    tonFollowerSeq: TON;
	FollowerSeq: SequenceTransfer;	
	lrPosCnt: INT;
	i: INT;
	bRecipeComplete: BOOL;
	rtMasterInRange: R_TRIG;
	bTriggerPos: BOOL;
	tonDelayMotion: TON;
END_VAR

VAR CONSTANT
	iCamID1: MC_CAM_ID:=4;	
    iCamID2: MC_CAM_ID:=5;		
END_VAR

//减速比10/1 同步轮周长400 ，皮带总长3300，7个工位，工位间距60
Ref_MachineStateModel REF= UN01_MachineStateModel;
Ref_Unit REF=Unit01;
ref_Master REF= arVirtualAxisAdmin[1];
ref_Follower1  REF= arRealAxisAdmin[44];
ref_Follower2  REF= arRealAxisAdmin[45];
MainRoution();
CM01_Cam1();
CM02_Cam2();

ACTION Cam1Table:
//凸轮1曲线
camTableFollower1.ArraySize:=SIZEOF(table1);
camTableFollower1.NoOfColumns:=1;
camTableFollower1.NoOfRows:=13;
camTableFollower1.pArray:=ADR(table1);
camTableFollower1.TableType:=MC_TABLETYPE_MOTIONFUNCTION;

{region Table}

//0
table1[1].FunctionType:=MOTIONFUNCTYPE_POLYNOM5;
table1[1].MasterPos:=0;
table1[1].SlavePos:=0;
table1[1].PointIndex:=1;
table1[1].PointType:=MOTIONPOINTTYPE_MOTION;

//1	 (dist200)
table1[2].FunctionType:=MOTIONFUNCTYPE_POLYNOM5;
table1[2].MasterPos:=200;
table1[2].SlavePos:=80;
table1[2].PointIndex:=2;
table1[2].PointType:=MOTIONPOINTTYPE_MOTION;
//2   (dist200)
table1[3].FunctionType:=MOTIONFUNCTYPE_POLYNOM5;
table1[3].MasterPos:=400;
table1[3].SlavePos:=table1[2].SlavePos+60;
table1[3].PointIndex:=3;
table1[3].PointType:=MOTIONPOINTTYPE_MOTION;
//3   (dist200)
table1[4].FunctionType:=MOTIONFUNCTYPE_POLYNOM5;
table1[4].MasterPos:=600;
table1[4].SlavePos:=table1[3].SlavePos+60;
table1[4].PointIndex:=4;
table1[4].PointType:=MOTIONPOINTTYPE_MOTION;
//4  (dist200)
table1[5].FunctionType:=MOTIONFUNCTYPE_POLYNOM5;
table1[5].MasterPos:=800;
table1[5].SlavePos:=table1[4].SlavePos+60;
table1[5].PointIndex:=5;
table1[5].PointType:=MOTIONPOINTTYPE_MOTION;
//5  (dist200)
table1[6].FunctionType:=MOTIONFUNCTYPE_POLYNOM5;
table1[6].MasterPos:=1000;
table1[6].SlavePos:=table1[5].SlavePos+60;
table1[6].PointIndex:=6;
table1[6].PointType:=MOTIONPOINTTYPE_MOTION;
//6  (dist200)
table1[7].FunctionType:=MOTIONFUNCTYPE_POLYNOM5;
table1[7].MasterPos:=1200;
table1[7].SlavePos:=table1[6].SlavePos+60;
table1[7].PointIndex:=7;
table1[7].PointType:=MOTIONPOINTTYPE_MOTION;
//7  (dist200)
table1[8].FunctionType:=MOTIONFUNCTYPE_POLYNOM5;
table1[8].MasterPos:=1400;
table1[8].SlavePos:=table1[7].SlavePos+60;
table1[8].PointIndex:=8;
table1[8].PointType:=MOTIONPOINTTYPE_MOTION;
//900   (dist0)
table1[9].FunctionType:=MOTIONFUNCTYPE_POLYNOM5;
table1[9].MasterPos:=1600;
table1[9].SlavePos:=table1[8].SlavePos+900;
table1[9].PointIndex:=9;
table1[9].PointType:=MOTIONPOINTTYPE_MOTION;
//900  (dist0)
table1[10].FunctionType:=MOTIONFUNCTYPE_POLYNOM5;
table1[10].MasterPos:=1800;
table1[10].SlavePos:=table1[9].SlavePos;
table1[10].PointIndex:=10;
table1[10].PointType:=MOTIONPOINTTYPE_MOTION;
//900  (dist0)
table1[11].FunctionType:=MOTIONFUNCTYPE_POLYNOM5;
table1[11].MasterPos:=2000;
table1[11].SlavePos:=table1[10].SlavePos;
table1[11].PointIndex:=11;
table1[11].PointType:=MOTIONPOINTTYPE_MOTION;
//3240 (dist700)
table1[12].FunctionType:=MOTIONFUNCTYPE_POLYNOM1;
table1[12].MasterPos:=2700;
table1[12].SlavePos:= 3240;
table1[12].PointIndex:=12;
table1[12].PointType:=MOTIONPOINTTYPE_MOTION;
//3300 (dist100)
table1[13].FunctionType:=MOTIONFUNCTYPE_POLYNOM5;
table1[13].MasterPos:=2800;
table1[13].SlavePos:=3300;
table1[13].PointIndex:=13;
table1[13].PointType:=MOTIONPOINTTYPE_MOTION;

{endRegion}
END_ACTION

ACTION Cam1Table_1:
//凸轮1曲线
camTableFollower1.ArraySize:=SIZEOF(table1);
camTableFollower1.NoOfColumns:=1;
camTableFollower1.NoOfRows:=27;
camTableFollower1.pArray:=ADR(table1);
camTableFollower1.TableType:=MC_TABLETYPE_MOTIONFUNCTION;

{region Table}

//0
table1[1].FunctionType:=MOTIONFUNCTYPE_POLYNOM5;
table1[1].MasterPos:=0;
table1[1].SlavePos:=0;
table1[1].PointIndex:=1;
table1[1].PointType:=MOTIONPOINTTYPE_MOTION;

//1	 (dist200)
table1[2].FunctionType:=MOTIONFUNCTYPE_POLYNOM5;
table1[2].MasterPos:=20;
table1[2].SlavePos:=0;
table1[2].PointIndex:=2;
table1[2].PointType:=MOTIONPOINTTYPE_MOTION;

//1	 (dist200)
table1[3].FunctionType:=MOTIONFUNCTYPE_POLYNOM5;
table1[3].MasterPos:=100;
table1[3].SlavePos:=80;
table1[3].PointIndex:=3;
table1[3].PointType:=MOTIONPOINTTYPE_MOTION;
	 
//1	 (dist200)
table1[4].FunctionType:=MOTIONFUNCTYPE_POLYNOM5;
table1[4].MasterPos:=200;
table1[4].SlavePos:=80;
table1[4].PointIndex:=4;
table1[4].PointType:=MOTIONPOINTTYPE_MOTION;
		  
//2   (dist200)
table1[5].FunctionType:=MOTIONFUNCTYPE_POLYNOM5;
table1[5].MasterPos:=220;
table1[5].SlavePos:=80;
table1[5].PointIndex:=5;
table1[5].PointType:=MOTIONPOINTTYPE_MOTION;

//2   (dist200)
table1[6].FunctionType:=MOTIONFUNCTYPE_POLYNOM5;
table1[6].MasterPos:=300;
table1[6].SlavePos:=140;
table1[6].PointIndex:=6;
table1[6].PointType:=MOTIONPOINTTYPE_MOTION;
	 
//2   (dist200)
table1[7].FunctionType:=MOTIONFUNCTYPE_POLYNOM5;
table1[7].MasterPos:=400;
table1[7].SlavePos:=140;
table1[7].PointIndex:=7;
table1[7].PointType:=MOTIONPOINTTYPE_MOTION;

//3   (dist200)
table1[8].FunctionType:=MOTIONFUNCTYPE_POLYNOM5;
table1[8].MasterPos:=420;
table1[8].SlavePos:=200;
table1[8].PointIndex:=8;
table1[8].PointType:=MOTIONPOINTTYPE_MOTION;
		  
//3   (dist200)
table1[9].FunctionType:=MOTIONFUNCTYPE_POLYNOM5;
table1[9].MasterPos:=500;
table1[9].SlavePos:=200;
table1[9].PointIndex:=9;
table1[9].PointType:=MOTIONPOINTTYPE_MOTION;
	 
//3   (dist200)
table1[10].FunctionType:=MOTIONFUNCTYPE_POLYNOM5;
table1[10].MasterPos:=600;
table1[10].SlavePos:=200;
table1[10].PointIndex:=10;
table1[10].PointType:=MOTIONPOINTTYPE_MOTION;		  

//4  (dist200)
table1[11].FunctionType:=MOTIONFUNCTYPE_POLYNOM5;
table1[11].MasterPos:=620;
table1[11].SlavePos:=200;
table1[11].PointIndex:=11;
table1[11].PointType:=MOTIONPOINTTYPE_MOTION;
			   											 
//4  (dist200)
table1[12].FunctionType:=MOTIONFUNCTYPE_POLYNOM5;
table1[12].MasterPos:=700;
table1[12].SlavePos:=260;
table1[12].PointIndex:=12;
table1[12].PointType:=MOTIONPOINTTYPE_MOTION;
	 
//4  (dist200)
table1[13].FunctionType:=MOTIONFUNCTYPE_POLYNOM5;
table1[13].MasterPos:=800;
table1[13].SlavePos:=260;
table1[13].PointIndex:=13;
table1[13].PointType:=MOTIONPOINTTYPE_MOTION;		  
			 
//5  (dist200)
table1[14].FunctionType:=MOTIONFUNCTYPE_POLYNOM5;
table1[14].MasterPos:=820;
table1[14].SlavePos:=260;
table1[14].PointIndex:=14;
table1[14].PointType:=MOTIONPOINTTYPE_MOTION;
  				
//5  (dist200)
table1[15].FunctionType:=MOTIONFUNCTYPE_POLYNOM5;
table1[15].MasterPos:=900;
table1[15].SlavePos:=320;
table1[15].PointIndex:=15;
table1[15].PointType:=MOTIONPOINTTYPE_MOTION;
	 
//5  (dist200)
table1[16].FunctionType:=MOTIONFUNCTYPE_POLYNOM5;
table1[16].MasterPos:=1000;
table1[16].SlavePos:=320;
table1[16].PointIndex:=16;
table1[16].PointType:=MOTIONPOINTTYPE_MOTION;		  
	
//6  (dist200)
table1[17].FunctionType:=MOTIONFUNCTYPE_POLYNOM5;
table1[17].MasterPos:=1020;
table1[17].SlavePos:=320;
table1[17].PointIndex:=17;
table1[17].PointType:=MOTIONPOINTTYPE_MOTION;
		   						  							   
//6  (dist200)
table1[18].FunctionType:=MOTIONFUNCTYPE_POLYNOM5;
table1[18].MasterPos:=1100;
table1[18].SlavePos:=380;
table1[18].PointIndex:=18;
table1[18].PointType:=MOTIONPOINTTYPE_MOTION;
	 
//6  (dist200)
table1[19].FunctionType:=MOTIONFUNCTYPE_POLYNOM5;
table1[19].MasterPos:=1200;
table1[19].SlavePos:=380;
table1[19].PointIndex:=19;
table1[19].PointType:=MOTIONPOINTTYPE_MOTION;		  
	
//7  (dist200)
table1[20].FunctionType:=MOTIONFUNCTYPE_POLYNOM5;
table1[20].MasterPos:=1220;
table1[20].SlavePos:=380;
table1[20].PointIndex:=20;
table1[20].PointType:=MOTIONPOINTTYPE_MOTION;
							 										
//7  (dist200)
table1[21].FunctionType:=MOTIONFUNCTYPE_POLYNOM5;
table1[21].MasterPos:=1300;
table1[21].SlavePos:=440;
table1[21].PointIndex:=21;
table1[21].PointType:=MOTIONPOINTTYPE_MOTION;
	 
//7  (dist200)
table1[22].FunctionType:=MOTIONFUNCTYPE_POLYNOM5;
table1[22].MasterPos:=1400;
table1[22].SlavePos:=440;
table1[22].PointIndex:=22;
table1[22].PointType:=MOTIONPOINTTYPE_MOTION;		  
			   			 
//900   (dist900)
table1[23].FunctionType:=MOTIONFUNCTYPE_POLYNOM5;
table1[23].MasterPos:=1600;
table1[23].SlavePos:=440+900;
table1[23].PointIndex:=23;
table1[23].PointType:=MOTIONPOINTTYPE_MOTION;
//900  (dist0)
table1[24].FunctionType:=MOTIONFUNCTYPE_POLYNOM5;
table1[24].MasterPos:=1900;
table1[24].SlavePos:=1340;
table1[24].PointIndex:=24;
table1[24].PointType:=MOTIONPOINTTYPE_MOTION;
//900  (dist1860)
table1[25].FunctionType:=MOTIONFUNCTYPE_POLYNOM5;
table1[25].MasterPos:=2600;
table1[25].SlavePos:=3200;
table1[25].PointIndex:=25;
table1[25].PointType:=MOTIONPOINTTYPE_MOTION;
//3240 (dist40)
table1[26].FunctionType:=MOTIONFUNCTYPE_POLYNOM1;
table1[26].MasterPos:=2700;
table1[26].SlavePos:= 3240;
table1[26].PointIndex:=26;
table1[26].PointType:=MOTIONPOINTTYPE_MOTION;
//3300 (dist100)
table1[27].FunctionType:=MOTIONFUNCTYPE_POLYNOM5;
table1[27].MasterPos:=2800;
table1[27].SlavePos:=3300;
table1[27].PointIndex:=27;
table1[27].PointType:=MOTIONPOINTTYPE_MOTION;

{endRegion}
END_ACTION

ACTION Cam1Table_2:
//凸轮1曲线
camTableFollower1.ArraySize:=SIZEOF(table1);
camTableFollower1.NoOfColumns:=1;
camTableFollower1.NoOfRows:=20;
camTableFollower1.pArray:=ADR(table1);
camTableFollower1.TableType:=MC_TABLETYPE_MOTIONFUNCTION;

{region Table}

//0
table1[1].FunctionType:=MOTIONFUNCTYPE_POLYNOM5;
table1[1].MasterPos:=0;
table1[1].SlavePos:=0;
table1[1].PointIndex:=1;
table1[1].PointType:=MOTIONPOINTTYPE_MOTION;

//1	 (dist200)
table1[2].FunctionType:=MOTIONFUNCTYPE_POLYNOM5;
table1[2].MasterPos:=100;
table1[2].SlavePos:=80;
table1[2].PointIndex:=2;
table1[2].PointType:=MOTIONPOINTTYPE_MOTION;
	 
//1	 (dist200)
table1[3].FunctionType:=MOTIONFUNCTYPE_POLYNOM5;
table1[3].MasterPos:=200;
table1[3].SlavePos:=80;
table1[3].PointIndex:=3;
table1[3].PointType:=MOTIONPOINTTYPE_MOTION;
		  
//2   (dist200)
table1[4].FunctionType:=MOTIONFUNCTYPE_POLYNOM5;
table1[4].MasterPos:=300;
table1[4].SlavePos:=140;
table1[4].PointIndex:=4;
table1[4].PointType:=MOTIONPOINTTYPE_MOTION;
	 
//2   (dist200)
table1[5].FunctionType:=MOTIONFUNCTYPE_POLYNOM5;
table1[5].MasterPos:=400;
table1[5].SlavePos:=140;
table1[5].PointIndex:=5;
table1[5].PointType:=MOTIONPOINTTYPE_MOTION;

		  
//3   (dist200)
table1[6].FunctionType:=MOTIONFUNCTYPE_POLYNOM5;
table1[6].MasterPos:=500;
table1[6].SlavePos:=200;
table1[6].PointIndex:=6;
table1[6].PointType:=MOTIONPOINTTYPE_MOTION;
	 
//3   (dist200)
table1[7].FunctionType:=MOTIONFUNCTYPE_POLYNOM5;
table1[7].MasterPos:=600;
table1[7].SlavePos:=200;
table1[7].PointIndex:=7;
table1[7].PointType:=MOTIONPOINTTYPE_MOTION;		  
			   											 
//4  (dist200)
table1[8].FunctionType:=MOTIONFUNCTYPE_POLYNOM5;
table1[8].MasterPos:=700;
table1[8].SlavePos:=260;
table1[8].PointIndex:=8;
table1[8].PointType:=MOTIONPOINTTYPE_MOTION;
	 
//4  (dist200)
table1[9].FunctionType:=MOTIONFUNCTYPE_POLYNOM5;
table1[9].MasterPos:=800;
table1[9].SlavePos:=260;
table1[9].PointIndex:=9;
table1[9].PointType:=MOTIONPOINTTYPE_MOTION;		  
			   				
//5  (dist200)
table1[10].FunctionType:=MOTIONFUNCTYPE_POLYNOM5;
table1[10].MasterPos:=900;
table1[10].SlavePos:=320;
table1[10].PointIndex:=10;
table1[10].PointType:=MOTIONPOINTTYPE_MOTION;
	 
//5  (dist200)
table1[11].FunctionType:=MOTIONFUNCTYPE_POLYNOM5;
table1[11].MasterPos:=1000;
table1[11].SlavePos:=320;
table1[11].PointIndex:=11;
table1[11].PointType:=MOTIONPOINTTYPE_MOTION;		  
			   						  							   
//6  (dist200)
table1[12].FunctionType:=MOTIONFUNCTYPE_POLYNOM5;
table1[12].MasterPos:=1100;
table1[12].SlavePos:=380;
table1[12].PointIndex:=12;
table1[12].PointType:=MOTIONPOINTTYPE_MOTION;
	 
//6  (dist200)
table1[13].FunctionType:=MOTIONFUNCTYPE_POLYNOM5;
table1[13].MasterPos:=1200;
table1[13].SlavePos:=380;
table1[13].PointIndex:=13;
table1[13].PointType:=MOTIONPOINTTYPE_MOTION;		  
								 										
//7  (dist200)
table1[14].FunctionType:=MOTIONFUNCTYPE_POLYNOM5;
table1[14].MasterPos:=1300;
table1[14].SlavePos:=440;
table1[14].PointIndex:=14;
table1[14].PointType:=MOTIONPOINTTYPE_MOTION;
	 
//7  (dist200)
table1[15].FunctionType:=MOTIONFUNCTYPE_POLYNOM5;
table1[15].MasterPos:=1400;
table1[15].SlavePos:=440;
table1[15].PointIndex:=15;
table1[15].PointType:=MOTIONPOINTTYPE_MOTION;		  
			   			 
//900   (dist900)
table1[16].FunctionType:=MOTIONFUNCTYPE_POLYNOM5;
table1[16].MasterPos:=1600;
table1[16].SlavePos:=440+900;
table1[16].PointIndex:=16;
table1[16].PointType:=MOTIONPOINTTYPE_MOTION;
//900  (dist0)
table1[17].FunctionType:=MOTIONFUNCTYPE_POLYNOM5;
table1[17].MasterPos:=1900;
table1[17].SlavePos:=1340;
table1[17].PointIndex:=17;
table1[17].PointType:=MOTIONPOINTTYPE_MOTION;
//900  (dist1860)
table1[18].FunctionType:=MOTIONFUNCTYPE_POLYNOM5;
table1[18].MasterPos:=2600;
table1[18].SlavePos:=3200;
table1[18].PointIndex:=18;
table1[18].PointType:=MOTIONPOINTTYPE_MOTION;
//3240 (dist40)
table1[19].FunctionType:=MOTIONFUNCTYPE_POLYNOM1;
table1[19].MasterPos:=2700;
table1[19].SlavePos:= 3240;
table1[19].PointIndex:=19;
table1[19].PointType:=MOTIONPOINTTYPE_MOTION;
//3300 (dist100)
table1[20].FunctionType:=MOTIONFUNCTYPE_POLYNOM5;
table1[20].MasterPos:=2800;
table1[20].SlavePos:=3300;
table1[20].PointIndex:=20;
table1[20].PointType:=MOTIONPOINTTYPE_MOTION;

{endRegion}
END_ACTION

ACTION Cam2Table:
//凸轮2曲线
camTableFollower2.ArraySize:=SIZEOF(table2);
camTableFollower2.NoOfColumns:=1;
camTableFollower2.NoOfRows:=13;
camTableFollower2.pArray:=ADR(table2);
camTableFollower2.TableType:=MC_TABLETYPE_MOTIONFUNCTION;

{region Table}
//7		 							  
table2[1].FunctionType:=MOTIONFUNCTYPE_POLYNOM5;
table2[1].MasterPos:=0;
table2[1].SlavePos:=0;
table2[1].PointIndex:=1;
table2[1].PointType:=MOTIONPOINTTYPE_MOTION;
//900	 (dist300)
table2[2].FunctionType:=MOTIONFUNCTYPE_POLYNOM5;
table2[2].MasterPos:=200;
table2[2].SlavePos:=900;
table2[2].PointIndex:=2;
table2[2].PointType:=MOTIONPOINTTYPE_MOTION;
//900    (dist0)
table2[3].FunctionType:=MOTIONFUNCTYPE_POLYNOM5;
table2[3].MasterPos:=400;
table2[3].SlavePos:=table2[2].SlavePos;
table2[3].PointIndex:=3;
table2[3].PointType:=MOTIONPOINTTYPE_MOTION;
//900    (dist0)
table2[4].FunctionType:=MOTIONFUNCTYPE_POLYNOM5;
table2[4].MasterPos:=600;
table2[4].SlavePos:=table2[3].SlavePos;
table2[4].PointIndex:=4;
table2[4].PointType:=MOTIONPOINTTYPE_MOTION;
//2800 (dist 700)
table2[5].FunctionType:=MOTIONFUNCTYPE_POLYNOM1;
table2[5].MasterPos:=1300;
table2[5].SlavePos:=2800;
table2[5].PointIndex:=5;
table2[5].PointType:=MOTIONPOINTTYPE_MOTION;
//2860 (dist 100)
table2[6].FunctionType:=MOTIONFUNCTYPE_POLYNOM1;
table2[6].MasterPos:=1400;
table2[6].SlavePos:=2860;
table2[6].PointIndex:=6;
table2[6].PointType:=MOTIONPOINTTYPE_MOTION;
//1 (dist 200)
table2[7].FunctionType:=MOTIONFUNCTYPE_POLYNOM5;
table2[7].MasterPos:=1600;
table2[7].SlavePos:=table2[6].SlavePos+80;
table2[7].PointIndex:=7;
table2[7].PointType:=MOTIONPOINTTYPE_MOTION;
//2 (dist 200)
table2[8].FunctionType:=MOTIONFUNCTYPE_POLYNOM5;
table2[8].MasterPos:=1800;
table2[8].SlavePos:=table2[7].SlavePos+60;
table2[8].PointIndex:=8;
table2[8].PointType:=MOTIONPOINTTYPE_MOTION;
//3 (dist 200)
table2[9].FunctionType:=MOTIONFUNCTYPE_POLYNOM5;
table2[9].MasterPos:=2000;
table2[9].SlavePos:=table2[8].SlavePos+60;
table2[9].PointIndex:=9;
table2[9].PointType:=MOTIONPOINTTYPE_MOTION;
//4 (dist 200)
table2[10].FunctionType:=MOTIONFUNCTYPE_POLYNOM5;
table2[10].MasterPos:=2200;
table2[10].SlavePos:=table2[9].SlavePos+60;
table2[10].PointIndex:=10;
table2[10].PointType:=MOTIONPOINTTYPE_MOTION;
//5 (dist 200)
table2[11].FunctionType:=MOTIONFUNCTYPE_POLYNOM5;
table2[11].MasterPos:=2400;
table2[11].SlavePos:=table2[10].SlavePos+60;
table2[11].PointIndex:=11;
table2[11].PointType:=MOTIONPOINTTYPE_MOTION;
//6 (dist 200)
table2[12].FunctionType:=MOTIONFUNCTYPE_POLYNOM5;
table2[12].MasterPos:=2600;
table2[12].SlavePos:=table2[11].SlavePos+60;
table2[12].PointIndex:=12;
table2[12].PointType:=MOTIONPOINTTYPE_MOTION;
//7 (dist 200)
table2[13].FunctionType:=MOTIONFUNCTYPE_POLYNOM5;
table2[13].MasterPos:=2800;
table2[13].SlavePos:=3300;
table2[13].PointIndex:=13;
table2[13].PointType:=MOTIONPOINTTYPE_MOTION;

{endRegion}
END_ACTION

ACTION Cam2Table_1:
//凸轮2曲线
camTableFollower2.ArraySize:=SIZEOF(table2);
camTableFollower2.NoOfColumns:=1;
camTableFollower2.NoOfRows:=27;
camTableFollower2.pArray:=ADR(table2);
camTableFollower2.TableType:=MC_TABLETYPE_MOTIONFUNCTION;

{region Table}
//7		 							  
table2[1].FunctionType:=MOTIONFUNCTYPE_POLYNOM5;
table2[1].MasterPos:=0;
table2[1].SlavePos:=0;
table2[1].PointIndex:=1;
table2[1].PointType:=MOTIONPOINTTYPE_MOTION;
	 
//900	 (dist900)
table2[2].FunctionType:=MOTIONFUNCTYPE_POLYNOM5;
table2[2].MasterPos:=200;
table2[2].SlavePos:=900;
table2[2].PointIndex:=2;
table2[2].PointType:=MOTIONPOINTTYPE_MOTION;
	 
//900    (dist0)
table2[3].FunctionType:=MOTIONFUNCTYPE_POLYNOM5;
table2[3].MasterPos:=500;
table2[3].SlavePos:=900;
table2[3].PointIndex:=3;
table2[3].PointType:=MOTIONPOINTTYPE_MOTION;
//900    (dist1860)
table2[4].FunctionType:=MOTIONFUNCTYPE_POLYNOM5;
table2[4].MasterPos:=1200;
table2[4].SlavePos:=2760;
table2[4].PointIndex:=4;
table2[4].PointType:=MOTIONPOINTTYPE_MOTION;
	 
//2800 (dist 40)
table2[5].FunctionType:=MOTIONFUNCTYPE_POLYNOM1;
table2[5].MasterPos:=1300;
table2[5].SlavePos:=2800;
table2[5].PointIndex:=5;
table2[5].PointType:=MOTIONPOINTTYPE_MOTION;
	 
//2860 (dist 100)
table2[6].FunctionType:=MOTIONFUNCTYPE_POLYNOM1;
table2[6].MasterPos:=1400;
table2[6].SlavePos:=2860;
table2[6].PointIndex:=6;
table2[6].PointType:=MOTIONPOINTTYPE_MOTION;
	 
//1 (dist 200)
table2[7].FunctionType:=MOTIONFUNCTYPE_POLYNOM5;
table2[7].MasterPos:=1420;
table2[7].SlavePos:=2860;
table2[7].PointIndex:=7;
table2[7].PointType:=MOTIONPOINTTYPE_MOTION;		  
			   
//1 (dist 200)
table2[8].FunctionType:=MOTIONFUNCTYPE_POLYNOM5;
table2[8].MasterPos:=1500;
table2[8].SlavePos:=2940;
table2[8].PointIndex:=8;
table2[8].PointType:=MOTIONPOINTTYPE_MOTION;
	 
//1 (dist 200)
table2[9].FunctionType:=MOTIONFUNCTYPE_POLYNOM5;
table2[9].MasterPos:=1600;
table2[9].SlavePos:=2940;
table2[9].PointIndex:=9;
table2[9].PointType:=MOTIONPOINTTYPE_MOTION;

//2 (dist 200)
table2[10].FunctionType:=MOTIONFUNCTYPE_POLYNOM5;
table2[10].MasterPos:=1620;
table2[10].SlavePos:=2940;
table2[10].PointIndex:=10;
table2[10].PointType:=MOTIONPOINTTYPE_MOTION;
	 
//2 (dist 200)
table2[11].FunctionType:=MOTIONFUNCTYPE_POLYNOM5;
table2[11].MasterPos:=1700;
table2[11].SlavePos:=3000;
table2[11].PointIndex:=11;
table2[11].PointType:=MOTIONPOINTTYPE_MOTION;
	 
//2 (dist 200)
table2[12].FunctionType:=MOTIONFUNCTYPE_POLYNOM5;
table2[12].MasterPos:=1800;
table2[12].SlavePos:=3000;
table2[12].PointIndex:=12;
table2[12].PointType:=MOTIONPOINTTYPE_MOTION;
	
//3 (dist 200)
table2[13].FunctionType:=MOTIONFUNCTYPE_POLYNOM5;
table2[13].MasterPos:=1820;
table2[13].SlavePos:=3000;
table2[13].PointIndex:=13;
table2[13].PointType:=MOTIONPOINTTYPE_MOTION;
 
//3 (dist 200)
table2[14].FunctionType:=MOTIONFUNCTYPE_POLYNOM5;
table2[14].MasterPos:=1900;
table2[14].SlavePos:=3060;
table2[14].PointIndex:=14;
table2[14].PointType:=MOTIONPOINTTYPE_MOTION;
	 
//3 (dist 200)
table2[15].FunctionType:=MOTIONFUNCTYPE_POLYNOM5;
table2[15].MasterPos:=2000;
table2[15].SlavePos:=3060;
table2[15].PointIndex:=15;
table2[15].PointType:=MOTIONPOINTTYPE_MOTION;
	  
//4 (dist 200)
table2[16].FunctionType:=MOTIONFUNCTYPE_POLYNOM5;
table2[16].MasterPos:=2020;
table2[16].SlavePos:=3060;
table2[16].PointIndex:=16;
table2[16].PointType:=MOTIONPOINTTYPE_MOTION;
	 
//4 (dist 200)
table2[17].FunctionType:=MOTIONFUNCTYPE_POLYNOM5;
table2[17].MasterPos:=2100;
table2[17].SlavePos:=3120;
table2[17].PointIndex:=17;
table2[17].PointType:=MOTIONPOINTTYPE_MOTION;		  
			   
//4 (dist 200)
table2[18].FunctionType:=MOTIONFUNCTYPE_POLYNOM5;
table2[18].MasterPos:=2200;
table2[18].SlavePos:=3120;
table2[18].PointIndex:=18;
table2[18].PointType:=MOTIONPOINTTYPE_MOTION;
	 
//5 (dist 200)
table2[19].FunctionType:=MOTIONFUNCTYPE_POLYNOM5;
table2[19].MasterPos:=2220;
table2[19].SlavePos:=3120;
table2[19].PointIndex:=19;
table2[19].PointType:=MOTIONPOINTTYPE_MOTION;
	 
//5 (dist 200)
table2[20].FunctionType:=MOTIONFUNCTYPE_POLYNOM5;
table2[20].MasterPos:=2300;
table2[20].SlavePos:=3180;
table2[20].PointIndex:=20;
table2[20].PointType:=MOTIONPOINTTYPE_MOTION;
		  
//5 (dist 200)
table2[21].FunctionType:=MOTIONFUNCTYPE_POLYNOM5;
table2[21].MasterPos:=2400;
table2[21].SlavePos:=3180;
table2[21].PointIndex:=21;
table2[21].PointType:=MOTIONPOINTTYPE_MOTION;	 
	 
//6 (dist 200)
table2[22].FunctionType:=MOTIONFUNCTYPE_POLYNOM5;
table2[22].MasterPos:=2420;
table2[22].SlavePos:=3180;
table2[22].PointIndex:=22;
table2[22].PointType:=MOTIONPOINTTYPE_MOTION;
		  
//6 (dist 200)
table2[23].FunctionType:=MOTIONFUNCTYPE_POLYNOM5;
table2[23].MasterPos:=2500;
table2[23].SlavePos:=3240;
table2[23].PointIndex:=23;
table2[23].PointType:=MOTIONPOINTTYPE_MOTION;

//6 (dist 200)
table2[24].FunctionType:=MOTIONFUNCTYPE_POLYNOM5;
table2[24].MasterPos:=2600;
table2[24].SlavePos:=3240;
table2[24].PointIndex:=24;
table2[24].PointType:=MOTIONPOINTTYPE_MOTION;	 
		  	   
//7 (dist 200)
table2[25].FunctionType:=MOTIONFUNCTYPE_POLYNOM5;
table2[25].MasterPos:=2620;
table2[25].SlavePos:=3240;
table2[25].PointIndex:=25;
table2[25].PointType:=MOTIONPOINTTYPE_MOTION;

//7 (dist 200)
table2[26].FunctionType:=MOTIONFUNCTYPE_POLYNOM5;
table2[26].MasterPos:=2700;
table2[26].SlavePos:=3300;
table2[26].PointIndex:=26;
table2[26].PointType:=MOTIONPOINTTYPE_MOTION;	 
		  
//7 (dist 200)
table2[27].FunctionType:=MOTIONFUNCTYPE_POLYNOM5;
table2[27].MasterPos:=2800;
table2[27].SlavePos:=3300;
table2[27].PointIndex:=27;
table2[27].PointType:=MOTIONPOINTTYPE_MOTION;
	 
{endRegion}
END_ACTION

ACTION Cam2Table_2:
//凸轮2曲线
camTableFollower2.ArraySize:=SIZEOF(table2);
camTableFollower2.NoOfColumns:=1;
camTableFollower2.NoOfRows:=20;
camTableFollower2.pArray:=ADR(table2);
camTableFollower2.TableType:=MC_TABLETYPE_MOTIONFUNCTION;

{region Table}
//7		 							  
table2[1].FunctionType:=MOTIONFUNCTYPE_POLYNOM5;
table2[1].MasterPos:=0;
table2[1].SlavePos:=0;
table2[1].PointIndex:=1;
table2[1].PointType:=MOTIONPOINTTYPE_MOTION;
//900	 (dist900)
table2[2].FunctionType:=MOTIONFUNCTYPE_POLYNOM5;
table2[2].MasterPos:=200;
table2[2].SlavePos:=900;
table2[2].PointIndex:=2;
table2[2].PointType:=MOTIONPOINTTYPE_MOTION;
//900    (dist0)
table2[3].FunctionType:=MOTIONFUNCTYPE_POLYNOM5;
table2[3].MasterPos:=500;
table2[3].SlavePos:=900;
table2[3].PointIndex:=3;
table2[3].PointType:=MOTIONPOINTTYPE_MOTION;
//900    (dist1860)
table2[4].FunctionType:=MOTIONFUNCTYPE_POLYNOM5;
table2[4].MasterPos:=1200;
table2[4].SlavePos:=2760;
table2[4].PointIndex:=4;
table2[4].PointType:=MOTIONPOINTTYPE_MOTION;
//2800 (dist 40)
table2[5].FunctionType:=MOTIONFUNCTYPE_POLYNOM1;
table2[5].MasterPos:=1300;
table2[5].SlavePos:=2800;
table2[5].PointIndex:=5;
table2[5].PointType:=MOTIONPOINTTYPE_MOTION;
//2860 (dist 100)
table2[6].FunctionType:=MOTIONFUNCTYPE_POLYNOM1;
table2[6].MasterPos:=1400;
table2[6].SlavePos:=2860;
table2[6].PointIndex:=6;
table2[6].PointType:=MOTIONPOINTTYPE_MOTION;
//1 (dist 200)
table2[7].FunctionType:=MOTIONFUNCTYPE_POLYNOM5;
table2[7].MasterPos:=1500;
table2[7].SlavePos:=2940;
table2[7].PointIndex:=7;
table2[7].PointType:=MOTIONPOINTTYPE_MOTION;
//1 (dist 200)
table2[8].FunctionType:=MOTIONFUNCTYPE_POLYNOM5;
table2[8].MasterPos:=1600;
table2[8].SlavePos:=2940;
table2[8].PointIndex:=8;
table2[8].PointType:=MOTIONPOINTTYPE_MOTION;
	 
//2 (dist 200)
table2[9].FunctionType:=MOTIONFUNCTYPE_POLYNOM5;
table2[9].MasterPos:=1700;
table2[9].SlavePos:=3000;
table2[9].PointIndex:=9;
table2[9].PointType:=MOTIONPOINTTYPE_MOTION;
//2 (dist 200)
table2[10].FunctionType:=MOTIONFUNCTYPE_POLYNOM5;
table2[10].MasterPos:=1800;
table2[10].SlavePos:=3000;
table2[10].PointIndex:=10;
table2[10].PointType:=MOTIONPOINTTYPE_MOTION;
	 
//3 (dist 200)
table2[11].FunctionType:=MOTIONFUNCTYPE_POLYNOM5;
table2[11].MasterPos:=1900;
table2[11].SlavePos:=3060;
table2[11].PointIndex:=11;
table2[11].PointType:=MOTIONPOINTTYPE_MOTION;
//3 (dist 200)
table2[12].FunctionType:=MOTIONFUNCTYPE_POLYNOM5;
table2[12].MasterPos:=2000;
table2[12].SlavePos:=3060;
table2[12].PointIndex:=12;
table2[12].PointType:=MOTIONPOINTTYPE_MOTION;
	  
//4 (dist 200)
table2[13].FunctionType:=MOTIONFUNCTYPE_POLYNOM5;
table2[13].MasterPos:=2100;
table2[13].SlavePos:=3120;
table2[13].PointIndex:=13;
table2[13].PointType:=MOTIONPOINTTYPE_MOTION;
//4 (dist 200)
table2[14].FunctionType:=MOTIONFUNCTYPE_POLYNOM5;
table2[14].MasterPos:=2200;
table2[14].SlavePos:=3120;
table2[14].PointIndex:=14;
table2[14].PointType:=MOTIONPOINTTYPE_MOTION;
	 
//5 (dist 200)
table2[15].FunctionType:=MOTIONFUNCTYPE_POLYNOM5;
table2[15].MasterPos:=2300;
table2[15].SlavePos:=3180;
table2[15].PointIndex:=15;
table2[15].PointType:=MOTIONPOINTTYPE_MOTION;
//5 (dist 200)
table2[16].FunctionType:=MOTIONFUNCTYPE_POLYNOM5;
table2[16].MasterPos:=2400;
table2[16].SlavePos:=3180;
table2[16].PointIndex:=16;
table2[16].PointType:=MOTIONPOINTTYPE_MOTION;	 
	 
//6 (dist 200)
table2[17].FunctionType:=MOTIONFUNCTYPE_POLYNOM5;
table2[17].MasterPos:=2500;
table2[17].SlavePos:=3240;
table2[17].PointIndex:=17;
table2[17].PointType:=MOTIONPOINTTYPE_MOTION;

//6 (dist 200)
table2[18].FunctionType:=MOTIONFUNCTYPE_POLYNOM5;
table2[18].MasterPos:=2600;
table2[18].SlavePos:=3240;
table2[18].PointIndex:=18;
table2[18].PointType:=MOTIONPOINTTYPE_MOTION;	 
		  	   
//7 (dist 200)
table2[19].FunctionType:=MOTIONFUNCTYPE_POLYNOM5;
table2[19].MasterPos:=2700;
table2[19].SlavePos:=3300;
table2[19].PointIndex:=19;
table2[19].PointType:=MOTIONPOINTTYPE_MOTION;
//7 (dist 200)
table2[20].FunctionType:=MOTIONFUNCTYPE_POLYNOM5;
table2[20].MasterPos:=2800;
table2[20].SlavePos:=3300;
table2[20].PointIndex:=20;
table2[20].PointType:=MOTIONPOINTTYPE_MOTION;
	 
{endRegion}
END_ACTION

ACTION CM01_Cam1:
Cam1Table();
	 
MC_CamIn_Follower1.Scaling.MasterRelative:=FALSE;
MC_CamIn_Follower1.Scaling.SlaveRelative:=FALSE;	 
	 
MC_CamIn_Follower1(
	Master:=ref_Master.Axis , 
	Slave:= ref_Follower1.Axis, 
	Execute:= ref_Follower1.i.CamIn, 
	ActivationMode:= , 
	ActivationPosition:= , 
	CamTableID:=iCamID1 , 
	Scaling:= , 
	Options:= , 
	InSync=> ref_Follower1.o.InCam, 
	Busy=> , 
	Active=> , 
	CommandAborted=> , 
	Error=> , 
	ErrorID=> );	
	
MC_CamTableSelect_Follower1(
	Master:= ref_Master.Axis, 
	Slave:= ref_Follower1.Axis, 
	CamTable:= CamTableFollower1, 
	Execute:= ref_Follower1.i.SelectCamTable, 
	Periodic:= TRUE, 
	MasterAbsolute:= , 
	SlaveAbsolute:= , 
	CamTableID:= iCamID1, 
	Done=> ref_Follower1.o.SelectCamTableDone, 
	Busy=> , 
	Error=> , 
	ErrorID=> );


MC_GearIn_Follower1(
	Master:=ref_Follower2.Axis , 
	Slave:=ref_Follower1.Axis , 
	Execute:=ref_Follower1.i.GearIn , 
	RatioNumerator:= 1, 
	RatioDenominator:= 1, 
	Acceleration:= , 
	Deceleration:= , 
	Jerk:= , 
	BufferMode:= , 
	Options:= , 
	InGear=> ref_Follower1.o.InGear, 
	Busy=> , 
	Active=> , 
	CommandAborted=> , 
	Error=> , 
	ErrorID=> );	
	
MC_ReadCamTableSlaveDynamicsFollwer1(
	Execute:= , 
	CamTableID:= iCamID1, 
	MasterPosition:= ref_Master.o.ActPos, 
	Done=> , 
	Busy=> , 
	Error=> , 
	ErrorID=> , 
	SlavePosition=> , 
	SlaveVelocity=> , 
	SlaveAcceleration=> );
END_ACTION

ACTION CM02_Cam2:
Cam2Table();

MC_CamIn_Follower2.Scaling.MasterRelative:=FALSE;
MC_CamIn_Follower2.Scaling.SlaveRelative:=FALSE;		 
MC_CamIn_Follower2(
	Master:=ref_Master.Axis , 
	Slave:= ref_Follower2.Axis, 
	Execute:= ref_Follower2.i.CamIn, 
	ActivationMode:= , 
	ActivationPosition:= , 
	CamTableID:=iCamID2 , 
	Scaling:= , 
	Options:= , 
	InSync=> ref_Follower2.o.InCam, 
	Busy=> , 
	Active=> , 
	CommandAborted=> , 
	Error=> , 
	ErrorID=> );	
	
MC_CamTableSelect_Follower2(
	Master:= ref_Master.Axis, 
	Slave:= ref_Follower2.Axis, 
	CamTable:= CamTableFollower2, 
	Execute:= ref_Follower2.i.SelectCamTable, 
	Periodic:= TRUE, 
	MasterAbsolute:= , 
	SlaveAbsolute:= , 
	CamTableID:= iCamID2, 
	Done=> ref_Follower2.o.SelectCamTableDone, 
	Busy=> , 
	Error=> , 
	ErrorID=> );

MC_GearIn_Follower2(
	Master:=ref_Follower1.Axis , 
	Slave:=ref_Follower2.Axis , 
	Execute:=ref_Follower2.i.GearIn , 
	RatioNumerator:= 1, 
	RatioDenominator:= 1, 
	Acceleration:= , 
	Deceleration:= , 
	Jerk:= , 
	BufferMode:= , 
	Options:= , 
	InGear=> ref_Follower2.o.InGear, 
	Busy=> , 
	Active=> , 
	CommandAborted=> , 
	Error=> , 
	ErrorID=> );		
	
	
MC_ReadCamTableSlaveDynamicsFollwer2(
	Execute:= , 
	CamTableID:= iCamID2, 
	MasterPosition:= ref_Master.o.ActPos, 
	Done=> , 
	Busy=> , 
	Error=> , 
	ErrorID=> , 
	SlavePosition=> , 
	SlaveVelocity=> , 
	SlaveAcceleration=> );
END_ACTION

ACTION CM03_Follower:
CASE FollowerSeq.Now OF
	0: 
	   IF Ref_MachineStateModel.Sts_Resetting THEN
		  FollowerSeq(ExeCute:= TRUE, Next:= Seq_Resetting);  
	   END_IF	
	   IF Ref_MachineStateModel.Sts_Stopping  THEN
		  FollowerSeq(ExeCute:= TRUE, Next:= Seq_Stopping);  
	   END_IF
	   IF Ref_MachineStateModel.Sts_Execute  THEN
		  FollowerSeq(ExeCute:= TRUE, Next:= 110);   
	   END_IF
{region Resetting} 
	10:
		IF NOT ref_Follower1.o.PowerOn  THEN;
		   ref_Follower1.i.Enable:=TRUE;
		END_IF
		IF NOT ref_Follower2.o.PowerOn  THEN;
		   ref_Follower2.i.Enable:=TRUE;
		END_IF	
		
		IF ref_Follower1.o.PowerOn AND ref_Follower2.o.PowerOn THEN
		   FollowerSeq(ExeCute:= TRUE, Next:= 20);  
		END_IF
        IF Ref_MachineStateModel.Sts_Stopping  THEN
		   FollowerSeq(ExeCute:= TRUE, Next:= Seq_Stopping);  
	    END_IF	
		
	20:
		IF glb_AllAxisHomed_UN01 THEN
		   FollowerSeq(ExeCute:= TRUE, Next:= 21);
		   ELSE 
		   FollowerSeq(ExeCute:= TRUE, Next:= 30);
		END_IF
		
	21:
		IF ref_Master.o.Homed AND ref_Master.o.PowerOn THEN
		   FollowerSeq(ExeCute:= TRUE, Next:= 60);//轴组耦合
		END_IF
	30:
	   glb_lrMasterWrkCnt:=0;
	   glb_lrMasterTargetCnt:=0;
	   bRecipeComplete:=FALSE;
       MEMSET(destAddr:= ADR(glb_BinBelt4_5), fillByte:= 0, n:= SIZEOF(glb_BinBelt4_5));      
	   FollowerSeq(ExeCute:= TRUE, Next:= 40);
	
	40: 
	   ref_Follower1.i.GearIn:=TRUE;
	   IF ref_Follower1.o.InGear THEN
		  FollowerSeq(ExeCute:= TRUE, Next:= 41);
	   END_IF
	   
	41:
       ref_Follower2.i.HomeMode:=0;
       ref_Follower2.i.HomeOffset:=290;  //	
	   tonFollowerSeq(IN:=TRUE , PT:=T#1S , Q=> , ET=> );
	   IF tonFollowerSeq.Q THEN
		  tonFollowerSeq(IN:=FALSE , PT:=T#1S , Q=> , ET=> );	   
			ref_Follower2.i.Home:=TRUE;
			FollowerSeq(ExeCute:= TRUE, Next:= 42);
	   END_IF
	   
	42:
       IF ref_Follower2.o.HomeDone THEN
		  ref_Follower2.i.Home:=FALSE;
		  FollowerSeq(ExeCute:= TRUE, Next:= 43); 
	   ELSE IF Ref_MachineStateModel.Sts_Stopping  THEN
		       ref_Follower2.i.Home:=FALSE;
               FollowerSeq(ExeCute:= TRUE, Next:= Seq_Stopping);
	        END_IF
	   END_IF
	   
	43:
	   ref_Follower1.i.GearOut:=TRUE;
	   IF ref_Follower1.o.GearOutDone AND NOT ref_Follower1.o.InSync THEN
		  ref_Follower1.i.GearOut:=FALSE;
		  ref_Follower1.i.GearIn:=FALSE;
		  FollowerSeq(ExeCute:= TRUE, Next:= 44); 
	   END_IF
	   
	44:
	   IF ref_Follower1.o.StandStill THEN
          FollowerSeq(ExeCute:= TRUE, Next:= 45);
	   ELSE IF Ref_MachineStateModel.Sts_Stopping  THEN
		       FollowerSeq(ExeCute:= TRUE, Next:= Seq_Stopping);   
		    END_IF	  
	   END_IF
	   
	45:
	   ref_Follower2.i.GearIn:=TRUE;
	   IF ref_Follower2.o.InGear THEN
		  FollowerSeq(ExeCute:= TRUE, Next:= 46); 
	   END_IF  
	46:
	      ref_Follower1.i.HomeOffset:=290; // 
	      tonFollowerSeq(IN:=TRUE , PT:=T#1S , Q=> , ET=> );
	   IF tonFollowerSeq.Q THEN
			tonFollowerSeq(IN:=FALSE , PT:=T#1S , Q=> , ET=> );	   
			ref_Follower1.i.Home:=TRUE;
			FollowerSeq(ExeCute:= TRUE, Next:= 47); 
	   END_IF
	   
	47:
       IF ref_Follower1.o.HomeDone THEN
		   ref_Follower1.i.Home:=FALSE;
		   FollowerSeq(ExeCute:= TRUE, Next:= 48);
	   ELSE IF Ref_MachineStateModel.Sts_Stopping  THEN
		       ref_Follower1.i.Home:=FALSE;
               FollowerSeq(ExeCute:= TRUE, Next:= Seq_Stopping);   
		    END_IF 
	   END_IF
	48:
    	 ref_Follower1.i.Pos:=0 ; 
	     ref_Follower1.i.Vel:=100;
	     ref_Follower1.i.Acc:=600;
	     ref_Follower1.i.Dec:=600;   
		 FollowerSeq(ExeCute:= TRUE, Next:= 49);
    49: 
		 ref_Follower1.i.MoveAbs:=TRUE;
	     IF  ref_Follower1.o.CmdDone  THEN
			 ref_Follower1.i.MoveAbs:=FALSE; 
			 FollowerSeq(ExeCute:= TRUE, Next:= 50);
	     ELSE IF Ref_MachineStateModel.Sts_Stopping  THEN
		         ref_Follower1.i.MoveAbs:=FALSE;
                 FollowerSeq(ExeCute:= TRUE, Next:= Seq_Stopping);   
		      END_IF			 
		 END_IF
	      
	50:
	   ref_Follower2.i.GearOut:=TRUE;
	   IF ref_Follower2.o.GearOutDone  THEN
		  ref_Follower2.i.GearOut:=FALSE;
		  ref_Follower2.i.GearIn:=FALSE;
		  FollowerSeq(ExeCute:= TRUE, Next:= 51); 
	   END_IF  
	51: 
        tonFollowerSeq(IN:=TRUE , PT:=T#500MS , Q=> , ET=> );
		IF  ref_Follower2.o.StandStill AND tonFollowerSeq.Q  THEN
			 tonFollowerSeq(IN:=FALSE , PT:=T#500MS , Q=> , ET=> );
		     FollowerSeq(ExeCute:= TRUE, Next:= 52);
	    END_IF
		
	52: 
		 ref_Follower2.i.Dist:=440-ref_Follower2.o.ActPos ; 
         lrFollower2PosLast:=ref_Follower2.i.Pos;
	     ref_Follower2.i.Vel:=100;
	     ref_Follower2.i.Acc:=6000;
	     ref_Follower2.i.Dec:=600;
		 FollowerSeq(ExeCute:= TRUE, Next:= 53);
		 
    53:  ref_Follower2.i.MoveReal:=TRUE; 
		 FollowerSeq(ExeCute:= TRUE, Next:= 54);

    54:		 
         IF  ref_Follower2.o.CmdDone  THEN
			 ref_Follower2.i.MoveReal:=FALSE; 
			 FollowerSeq(ExeCute:= TRUE, Next:= 55);
	     ELSE IF Ref_MachineStateModel.Sts_Stopping  THEN
                 FollowerSeq(ExeCute:= TRUE, Next:= Seq_Stopping);    
		      END_IF			 
		 END_IF
    55: 		 
	   ref_Follower2.i.Home:=TRUE;
	   ref_Follower2.i.HomeOffset:=0;  
	   ref_Follower2.i.HomeMode:=2;
	   FollowerSeq(ExeCute:= TRUE, Next:= 56); 
	   
	56:
       IF ref_Follower2.o.HomeDone THEN
		   ref_Follower2.i.Home:=FALSE;
		   FollowerSeq(ExeCute:= TRUE, Next:= 60);  
	   ELSE IF Ref_MachineStateModel.Sts_Stopping  THEN
		       FollowerSeq(ExeCute:= TRUE, Next:= Seq_Stopping);   
		    END_IF		   
	   END_IF
	   
	60:
	   ref_Follower1.i.SelectCamTable:=TRUE; 
	   IF ref_Follower1.o.SelectCamTableDone THEN
		   ref_Follower1.i.SelectCamTable:=FALSE; 
		   FollowerSeq(ExeCute:= TRUE, Next:= 61);  
	   END_IF
	   
	61:
        MC_ReadCamTableSlaveDynamicsFollwer1.Execute:=TRUE;
	    IF MC_ReadCamTableSlaveDynamicsFollwer1.Done THEN
			lrFollow1CamDynPos:=MC_ReadCamTableSlaveDynamicsFollwer1.SlavePosition
            +TRUNC(ref_master.o.ActPos/2800)*3300;
			lrFollow1LatchPos:=ref_Follower1.o.ActPos;
			MC_ReadCamTableSlaveDynamicsFollwer1.Execute:=FALSE;
			FollowerSeq(ExeCute:= TRUE, Next:= 62); 
		END_IF  
	62:
		ref_Follower2.i.SelectCamTable:=TRUE; 
		IF ref_Follower2.o.SelectCamTableDone THEN
		   ref_Follower2.i.SelectCamTable:=FALSE; 
		   FollowerSeq(ExeCute:= TRUE, Next:= 63);  
		END_IF
	63:
        MC_ReadCamTableSlaveDynamicsFollwer2.Execute:=TRUE;
	    IF MC_ReadCamTableSlaveDynamicsFollwer2.Done THEN
			lrFollow2CamDynPos:=MC_ReadCamTableSlaveDynamicsFollwer2.SlavePosition
            +TRUNC(ref_master.o.ActPos/2800)*3300;
			lrFollow2LatchPos:=ref_Follower2.o.ActPos;
			MC_ReadCamTableSlaveDynamicsFollwer2.Execute:=FALSE;
			FollowerSeq(ExeCute:= TRUE, Next:= 64); 
		END_IF  
    64:
	    tonFollowerSeq(IN:= TRUE, PT:= T#1S, Q=> , ET=> );
		IF tonFollowerSeq.Q THEN
		   tonFollowerSeq(IN:= FALSE, PT:= T#1S, Q=> , ET=> );	
		   FollowerSeq(ExeCute:= TRUE, Next:= 70); 
		END_IF
		
    70:
		ref_Follower1.i.Pos:=lrFollow1CamDynPos;
        ref_Follower1.i.Vel:=60;
		ref_Follower1.i.Acc:=600;
		ref_Follower1.i.Dec:=600;
		
		ref_Follower2.i.Pos:=lrFollow2CamDynPos;
		ref_Follower2.i.Vel:=60;
		ref_Follower2.i.Acc:=600;
		ref_Follower2.i.Dec:=600;		
        FollowerSeq(ExeCute:= TRUE, Next:= 71);  
	71: 
	    tonFollowerSeq(IN:= TRUE, PT:= T#1S, Q=> , ET=> );
		IF tonFollowerSeq.Q THEN
		   tonFollowerSeq(IN:= FALSE, PT:= T#1S, Q=> , ET=> );	
		   FollowerSeq(ExeCute:= TRUE, Next:= 72); 	   
		END_IF	
	72:	
		ref_Follower2.i.MoveAbs:=TRUE;
		ref_Follower1.i.MoveAbs:=TRUE;
	    IF ref_Follower1.o.CmdDone AND ref_Follower1.o.StandStill
        AND ref_Follower2.o.CmdDone AND ref_Follower2.o.StandStill THEN
			ref_Follower1.i.MoveAbs:=FALSE;
			ref_Follower2.i.MoveAbs:=FALSE;
			FollowerSeq(ExeCute:= TRUE, Next:= 73); 
	    ELSE IF Ref_MachineStateModel.Sts_Stopping  THEN
				ref_Follower1.i.MoveAbs:=FALSE;
				ref_Follower2.i.MoveAbs:=FALSE;			   
				FollowerSeq(ExeCute:= TRUE, Next:= Seq_Stopping);   
			 END_IF			
		END_IF
		
			
	73:
	   ref_Follower1.i.CamIn:=TRUE;
       IF ref_Follower1.o.InSync  THEN
		  FollowerSeq(ExeCute:= TRUE, Next:= 74);  
	   END_IF 
    74: 
	   ref_Follower2.i.CamIn:=TRUE;
       IF ref_Follower2.o.InSync  THEN
		  FollowerSeq(ExeCute:= TRUE, Next:= 80);  
	   END_IF 
 
    80:
		IF glb_AllAxisHomed_UN01 THEN
		   FollowerSeq(ExeCute:= TRUE, Next:= 90);
		   ELSE 
		   FollowerSeq(ExeCute:= TRUE, Next:= 81);
		END_IF
	81:		
		IF ref_Master.o.Homed AND ref_Master.o.PowerOn THEN
		   FollowerSeq(ExeCute:= TRUE, Next:= 82);//轴组耦合
		END_IF
    82:	 			  
		lrPosCnt:=1;
		ref_Master.i.Pos:=200;
		ref_Master.i.Acc:=100;
		ref_Master.i.Dec:=100;
		glb_BinBelt4_5.bin[1].arDrop[1]:=TRUE;
		glb_BinBelt4_5.bin[1].arDrop[8]:=TRUE;
		FollowerSeq(ExeCute:= TRUE, Next:= 83);
			
	83:
		ref_Master.i.MoveAbs:=TRUE;
		IF ref_Master.o.CmdDone THEN
		   ref_Master.i.MoveAbs:=FALSE;
		   FollowerSeq(ExeCute:= TRUE,Hold:=FALSE, Next:= 90);
		END_IF				 
					  

    90:	
	   FollowerSeq(ExeCute:= TRUE, Next:= Seq_ResettingDone);
	

   	Seq_ResettingDone: 
         IF NOT Ref_MachineStateModel.Sts_Resetting THEN
			FollowerSeq(ExeCute:= TRUE, Next:= 0); 
		 END_IF	
			  
				   
						
{endregion}			  
{region Execute}
	110:   
	   FollowerSeq(ExeCute:=TRUE , Next:= 120); 
			
	120:	  
	   IF NOT glb_BinBelt4_5.bin[9].arDrop[8] 
	   AND NOT glb_BinBelt4_5.bin[1].arDrop[1] THEN
		   FollowerSeq(ExeCute:= TRUE, Next:= 121);  ;
	   END_IF
	   IF Ref_MachineStateModel.Sts_Stopping  THEN
		  FollowerSeq(ExeCute:= TRUE, Next:= Seq_Stopping);  
	   END_IF
	
    121:
		 tonDelayMotion(IN:= TRUE, PT:= T#800MS, Q=> , ET=> );
		 IF tonDelayMotion.Q THEN
            tonDelayMotion(IN:= FALSE, PT:= T#800MS, Q=> , ET=> );
			FollowerSeq(ExeCute:= TRUE, Next:= 130,hold:=FALSE); 	 
         END_IF	  
 		 			  
	130: 
        ref_Master.i.Pos:= ref_Master.i.Pos+200;
		ref_Master.i.Acc:=50;
		ref_Master.i.Dec:=100;
		ref_Master.i.Vel:=100;
        FollowerSeq(ExeCute:= TRUE,hold:=FALSE, Next:= 140);  
		
	140:  
 
		ref_Master.i.MoveAbs:=TRUE;
		IF ref_Master.o.CmdDone THEN
		   ref_Master.i.MoveAbs:=FALSE;
		   FollowerSeq(ExeCute:= TRUE,Hold:=FALSE, Next:= 150);
		END_IF

		IF  ref_Master.i.Pos - ref_Master.o.ActPos <90 AND NOT bTriggerPos  THEN
	       glb_BinBelt4_5.bin[1].arDrop[1]:=TRUE;
		   bTriggerPos:=TRUE;
	    END_IF
	  
	     
	150:           
          bTriggerPos:=FALSE;
          glb_lrMasterWrkCnt:=glb_lrMasterWrkCnt+1;
		  FOR i:=16 TO 1 BY -1 DO
			  glb_BinBelt4_5.bin[i]:= glb_BinBelt4_5.bin[i-1];
		  END_FOR
		  FOR i:=16 TO 2 BY -1 DO
			  glb_BinBelt4_5.bin[i].arDrop[1]:= FALSE;
		  END_FOR			   
	      glb_BinBelt4_5.bin[1].arDrop[8]:=TRUE;		
		  FollowerSeq(ExeCute:=TRUE ,Hold:=FALSE, Next:= 110); 	   
	   
				  
{endRegion}
	Seq_Stopping: 
       ref_Master.i.Enable:=FALSE; 
	   IF NOT ref_Master.o.PowerOn THEN
			  FollowerSeq(ExeCute:= TRUE, Next:= 901); 	   
	   END_IF
	   
    901: 
	    IF NOT ref_Follower1.o.StandStill AND NOT ref_Follower1.o.InSync THEN
			ref_Follower1.i.Stop:=TRUE;
		END_IF	
	    IF NOT ref_Follower2.o.StandStill AND NOT ref_Follower2.o.InSync THEN
			ref_Follower2.i.Stop:=TRUE;
		END_IF
	    IF ref_Follower1.o.StandStill AND ref_Follower2.o.StandStill THEN
		   ref_Follower1.i.Stop:=FALSE;
		   ref_Follower2.i.Stop:=FALSE;
           FollowerSeq(ExeCute:= TRUE, Next:= 902); 		 
		END_IF
		
    902: 	

		IF ref_Follower1.o.InGear THEN 
		   ref_Follower1.i.GearOut:=TRUE;	
		END_IF	
		IF ref_Follower2.o.InGear THEN 
		   ref_Follower2.i.GearOut:=TRUE;	
		END_IF
		   FollowerSeq(ExeCute:= TRUE, Next:= 903); 
	903:
	    IF ref_Follower1.o.InSync THEN 
		   ref_Follower1.i.CamOut:=TRUE;	
		END_IF	
		IF ref_Follower2.o.InSync THEN 
		   ref_Follower2.i.CamOut:=TRUE;	
		END_IF	
		FollowerSeq(ExeCute:= TRUE, Next:= 904); 
	904:	
	    tonFollowerSeqDelay(IN:=TRUE , PT:=T#1S , Q=> , ET=> );
		IF tonFollowerSeqDelay.Q THEN
			tonFollowerSeqDelay(IN:=FALSE , PT:=T#1S , Q=> , ET=> );
			FollowerSeq(ExeCute:= TRUE, Next:= Seq_StoppingDone); 
		END_IF
			
	Seq_StoppingDone:
	     ref_Master.i.Disable:=TRUE;
	     ref_Follower1.i.Disable:=TRUE;
		 ref_Follower2.i.Disable:=TRUE;
		 IF NOT Ref_MachineStateModel.Sts_Stopping THEN
			FollowerSeq(ExeCute:= TRUE, Next:= 0); 	
		 END_IF
END_CASE
rtMasterInRange(CLK:= (ref_Master.o.ActPos- ref_Master.i.Pos >110)	, Q=> ); 
FollowerSeq.Hold := FALSE;
END_ACTION

ACTION MainRoution:
EM_No:=6;
IF Ref_Unit.EM_Selected[EM_No] THEN
	IF Ref_MachineStateModel.Sts_Holding THEN
		Ref_Unit.EM_Holding_Done[EM_No]:=TRUE;
		ELSE
		Ref_Unit.EM_Holding_Done[EM_No]:=FALSE;
	END_IF
	IF Ref_MachineStateModel.Sts_UnHolding THEN
		Ref_Unit.EM_UnHolding_Done[EM_No]:=TRUE;
		ELSE
		Ref_Unit.EM_UnHolding_Done[EM_No]:=FALSE;
	END_IF
	
	IF Ref_MachineStateModel.Sts_Suspending THEN
		Ref_Unit.EM_Suspending_Done[EM_No]:=TRUE;
		ELSE
		Ref_Unit.EM_Suspending_Done[EM_No]:=FALSE;
	END_IF
	
	IF Ref_MachineStateModel.Sts_UnSuspending THEN
		Ref_Unit.EM_UnSuspending_Done[EM_No]:=TRUE;
		ELSE
		Ref_Unit.EM_UnSuspending_Done[EM_No]:=FALSE;
	END_IF

	IF Ref_MachineStateModel.Sts_Resetting  AND FollowerSeq.Now=Seq_ResettingDone THEN
	   Ref_Unit.EM_Resetting_Done[EM_No]:=TRUE;
       ELSE   
	   Ref_Unit.EM_Resetting_Done[EM_No]:=FALSE;
	END_IF
	
	IF Ref_MachineStateModel.Sts_Clearing THEN
	   Ref_Unit.EM_Clearing_Done[EM_No]:=TRUE;
	   ELSE
	   Ref_Unit.EM_Clearing_Done[EM_No]:=FALSE;
	END_IF
	

	IF Ref_MachineStateModel.Sts_Starting THEN
	   Ref_Unit.EM_Starting_Done[EM_No]:=TRUE;
	   ELSE
       Ref_Unit.EM_Starting_Done[EM_No]:=FALSE;
	END_IF
	
	IF Ref_MachineStateModel.Sts_Stopping AND FollowerSeq.Now=Seq_StoppingDone  THEN
	   Ref_Unit.EM_Stopping_Done[EM_No]:=TRUE;	
       ELSE  
	   Ref_Unit.EM_Stopping_Done[EM_No]:=FALSE;	
	END_IF

	IF Ref_MachineStateModel.Sts_Aborting THEN
		FollowerSeq(ExeCute:= TRUE, Next:= 0);

		IF ref_Follower1.o.InSync THEN
			ref_Follower1.i.CamOut:=TRUE;
			ref_Follower1.i.GearOut:=TRUE;
		ELSE IF NOT ref_Follower1.o.StandStill THEN
				ref_follower1.i.Stop:=TRUE;
				END_IF		   
		END_IF
		
		IF ref_Follower2.o.InSync THEN
			ref_Follower2.i.CamOut:=TRUE;
			ref_Follower2.i.GearOut:=TRUE;
		ELSE IF NOT ref_Follower2.o.StandStill THEN
			ref_follower2.i.Stop:=TRUE;
			END_IF		   
		END_IF		   
	   
		IF tonAbortingWatchDog.Q THEN 
			Ref_Unit.EM_Aborting_Done[EM_No]:=TRUE;
			ref_Follower1.i.Disable:=TRUE;
			ref_Follower2.i.Disable:=TRUE;
        END_IF
    ELSE
		Ref_Unit.EM_Aborting_Done[EM_No]:=FALSE;
	END_IF
	
	tonAbortingWatchDog(IN:= Ref_MachineStateModel.Sts_Aborting, PT:=T#3S , Q=> , ET=> );
	CM03_Follower();
ELSE
		FollowerSeq(ExeCute:= TRUE, Next:= 0);		
END_IF
END_ACTION

END_PROGRAM

// ---- POUs/PackMaL_UN01/EM07_Belt6.TcPOU
PROGRAM EM07_Belt6
VAR
	ref_Master: REFERENCE TO UDT_AXISADMIN;
	ref_Belt: REFERENCE TO UDT_AXISADMIN;
	ref_Puller: REFERENCE TO UDT_AXISADMIN;
	ref_Encoder: REFERENCE TO Axis_Ref;
	ref_WindMotor: REFERENCE TO UDT_directMotor;
	Ref_MachineStateModel: REFERENCE TO PackMlv3_StateModel;
	ref_Work_Recipe: REFERENCE TO UDT_Hmi_Output; //当前生产的配方反馈给触摸屏
	Ref_Unit: REFERENCE TO UDT_UnitAdmin;	
	ref_BinList: REFERENCE TO UDT_BINlist;
	ref_diBeltObjCnt: REFERENCE TO DINT;
	ref_diPullFlag:REFERENCE TO DINT;
	ref_diDropFlag:REFERENCE TO DINT;
	ref_diCutFlag:REFERENCE TO DINT;	
	ref_diSealFlag:REFERENCE TO DINT;
	ref_diTransferFlag:REFERENCE TO DINT;	
	ref_bTransferPut:REFERENCE TO BOOL;
	ref_diGoodFlag:REFERENCE TO DINT;	
	ref_diNogoodFlag:REFERENCE TO DINT;	
	
	InfeedCylinder: REFERENCE TO UDT_Cylinderadmin;	
	InfeedSensor1: REFERENCE TO UDT_Sensoradmin;	
	InfeedSensor2: REFERENCE TO UDT_Sensoradmin;
	InfeedSensor3: REFERENCE TO UDT_Sensoradmin;
	InfeedSensor4: REFERENCE TO UDT_Sensoradmin;
	InfeedSensor5: REFERENCE TO UDT_Sensoradmin;
	InfeedSensor6: REFERENCE TO UDT_Sensoradmin;
	InfeedSensor7: REFERENCE TO UDT_Sensoradmin;
	InfeedSensor8: REFERENCE TO UDT_Sensoradmin;
	InfeedSensor9: REFERENCE TO UDT_Sensoradmin;
	InfeedSensor10: REFERENCE TO UDT_Sensoradmin;
	InfeedSensor11: REFERENCE TO UDT_Sensoradmin;
	InfeedSensor12: REFERENCE TO UDT_Sensoradmin;
	InfeedSensor13: REFERENCE TO UDT_Sensoradmin;
	InfeedSensor14: REFERENCE TO UDT_Sensoradmin;
	
	PullCylinder1: REFERENCE TO UDT_Cylinderadmin;	
	PullCylinder2: REFERENCE TO UDT_Cylinderadmin;
	PullCylinder3: REFERENCE TO UDT_Cylinderadmin;
	PullCylinder4: REFERENCE TO UDT_Cylinderadmin;
	PullCylinder5: REFERENCE TO UDT_Cylinderadmin;
	PullCylinder6: REFERENCE TO UDT_Cylinderadmin;
	PullCylinder7: REFERENCE TO UDT_Cylinderadmin;

	Check1Cylinder: REFERENCE TO UDT_Cylinderadmin;
	Check1Sensor1: REFERENCE TO UDT_Sensoradmin;	
	Check1Sensor2: REFERENCE TO UDT_Sensoradmin;
	Check1Sensor3: REFERENCE TO UDT_Sensoradmin;
	Check1Sensor4: REFERENCE TO UDT_Sensoradmin;
	Check1Sensor5: REFERENCE TO UDT_Sensoradmin;
	Check1Sensor6: REFERENCE TO UDT_Sensoradmin;
	Check1Sensor7: REFERENCE TO UDT_Sensoradmin;

	
	PullVacuum1: REFERENCE TO UDT_Vacuumadmin;
	PullVacuum2: REFERENCE TO UDT_Vacuumadmin;
	PullVacuum3: REFERENCE TO UDT_Vacuumadmin;
	PullVacuum4: REFERENCE TO UDT_Vacuumadmin;
	PullVacuum5: REFERENCE TO UDT_Vacuumadmin;
	PullVacuum6: REFERENCE TO UDT_Vacuumadmin;
	PullVacuum7: REFERENCE TO UDT_Vacuumadmin;	
	
	DropCylinderUP: REFERENCE TO UDT_Cylinderadmin;
	DropCylinderDown: REFERENCE TO UDT_Cylinderadmin;
	CutCylinderUP: REFERENCE TO UDT_Cylinderadmin;
	CutCylinderDown: REFERENCE TO UDT_Cylinderadmin;
	
    SealCylinderUP: REFERENCE TO UDT_Cylinderadmin;
    SealCylinderDown: REFERENCE TO UDT_Cylinderadmin;

    Seal2CylinderUP: REFERENCE TO UDT_Cylinderadmin;
    Seal2CylinderDown: REFERENCE TO UDT_Cylinderadmin;
	
    TransferCyliderHori: REFERENCE TO UDT_Cylinderadmin;
	TransferCyliderVert: REFERENCE TO UDT_Cylinderadmin;
	TransferCyliderRota: REFERENCE TO UDT_Cylinderadmin;
	
	TransferVacuum1: REFERENCE TO UDT_Vacuumadmin;
	TransferVacuum2: REFERENCE TO UDT_Vacuumadmin;
	TransferVacuum3: REFERENCE TO UDT_Vacuumadmin;
	TransferVacuum4: REFERENCE TO UDT_Vacuumadmin;
	TransferVacuum5: REFERENCE TO UDT_Vacuumadmin;
	TransferVacuum6: REFERENCE TO UDT_Vacuumadmin;
	TransferVacuum7: REFERENCE TO UDT_Vacuumadmin;	
	
	
	RejectCylinder: REFERENCE TO UDT_Cylinderadmin;
	
	
	
	EM_No: INT:=7;
	tonAbortingWatchDog: TON;

	tonDropSeq: ton;
	tonPullSeq: ton;	
	i: INT;
  
	tonTransferSeq: TON;
	tonSealSeq:  ton;
	tonSeal2Seq:  ton;
	IN: INT;
	bValveInitDone: BOOL;
	lrEncoderPosOld: LREAL;
	lrPosCnt: LREAL;
	tonBeltSeq: Ton;
	
	iValid: INT;
	rtTest: R_trig;
	bTestrt: BOOL;

	bBeltMove: BOOL;
	lrLatchMasterPos: LREAL;
	j: INT;
		
   
	PullSeq: SequenceTransfer;	
	DropSeq: SequenceTransfer;
	SealSeq: SequenceTransfer;
	Seal2Seq: SequenceTransfer;
	Check1Seq: SequenceTransfer;
	RejectSeq: SequenceTransfer;	
	CutSeq: SequenceTransfer;
	TransferSeq: SequenceTransfer;
	BeltSeq: SequenceTransfer;
	iTest: INT;
	lrTestPos: LREAL;
	tonCutSeq: TON;
	bBoxSealView: BOOL;
	bTestUpdata: BOOL;
	iBox: INT;
	iAutoCut: INT;
	tonCheck1Seq: Ton;
	tonRejectSeq: Ton;
	bRejectActive: BOOL;
END_VAR

VAR CONSTANT	
END_VAR
VAR RETAIN

END_VAR

//减速比50/1 同步轮周长57*15.875= 904.875，皮带总长462*15.875，33个工位，工位间距222.25
Ref_MachineStateModel REF= UN01_MachineStateModel;
Ref_Unit REF=Unit01;
ref_Master REF= arVirtualAxisAdmin[1];
ref_Belt REF= arRealAxisAdmin[46];
ref_Puller REF= arRealAxisAdmin[47];
ref_Work_Recipe REF=HMI_Output;
ref_diBeltObjCnt REF=glb_diBeltObjCnt;

ref_diPullFlag REF= glb_diPullFlag_UN01;
ref_diDropFlag REF= glb_diDropFlag_UN01;
ref_diCutFlag REF= glb_diCutFlag_UN01;
ref_diSealFlag REF= glb_diSealFlag_UN01;
ref_diGoodFlag REF= glb_diGoodFlag_UN01;
ref_diNogoodFlag REF= glb_diNogoodFlag_UN01;

ref_diTransferFlag REF= glb_diTransferFlag_UN01;
ref_bTransferPut REF= glb_bTransferPut_UN02;//

ref_Encoder REF= EncoderAxis[1];
ref_BinList REF=Glb_BinList;
ref_WindMotor REF= arPackMotor[1];
InfeedSensor1 REF= arPackSensor[1];
InfeedSensor2 REF= arPackSensor[2];
InfeedSensor3 REF= arPackSensor[3];
InfeedSensor4 REF= arPackSensor[4];
InfeedSensor5 REF= arPackSensor[5];
InfeedSensor6 REF= arPackSensor[6];
InfeedSensor7 REF= arPackSensor[7];
InfeedSensor8 REF= arPackSensor[8];
InfeedSensor9 REF= arPackSensor[9];
InfeedSensor10 REF= arPackSensor[10];
InfeedSensor11 REF= arPackSensor[11];
InfeedSensor12 REF= arPackSensor[12];
InfeedSensor13 REF= arPackSensor[13];
InfeedSensor14 REF= arPackSensor[14];

InfeedCylinder REF= arPackCylinder[9];
PullCylinder1 REF= arPackCylinder[1];
PullCylinder2 REF= arPackCylinder[2];
PullCylinder3 REF= arPackCylinder[3];
PullCylinder4 REF= arPackCylinder[4];
PullCylinder5 REF= arPackCylinder[5];
PullCylinder6 REF= arPackCylinder[6];
PullCylinder7 REF= arPackCylinder[7];

arPackCylinder[1].i.OutSensor:=TRUE;
arPackCylinder[2].i.OutSensor:=TRUE;
arPackCylinder[3].i.OutSensor:=TRUE;
arPackCylinder[4].i.OutSensor:=TRUE;
arPackCylinder[5].i.OutSensor:=TRUE;
arPackCylinder[6].i.OutSensor:=TRUE;
arPackCylinder[7].i.OutSensor:=TRUE;


DropCylinderUP REF= arPackCylinder[8];
DropCylinderDown REF= arPackCylinder[12];
DropCylinderDown.i.OutSensor:=TRUE;
CutCylinderUP REF= arPackCylinder[17];
CutCylinderDown REF= arPackCylinder[15];
TransferCyliderHori REF= arPackCylinder[14];
TransferCyliderVert REF= arPackCylinder[16];
TransferCyliderRota REF= arPackCylinder[13];

SealCylinderUP REF= arPackCylinder[10];
SealCylinderDown REF= arPackCylinder[11];

Seal2CylinderUP REF= arPackCylinder[18];
Seal2CylinderDown REF= arPackCylinder[19];

RejectCylinder REF= arPackCylinder[20];
RejectCylinder.i.InSensor:=TRUE;
RejectCylinder.i.OutSensor:=TRUE;

PullVacuum1 REF=arPackVacuum[1];
PullVacuum2 REF=arPackVacuum[2];
PullVacuum3 REF=arPackVacuum[3];
PullVacuum4 REF=arPackVacuum[4];
PullVacuum5 REF=arPackVacuum[5];
PullVacuum6 REF=arPackVacuum[6];
PullVacuum7 REF=arPackVacuum[7];

TransferVacuum1 REF=arPackVacuum[11];
TransferVacuum2 REF=arPackVacuum[12];
TransferVacuum3 REF=arPackVacuum[13];
TransferVacuum4 REF=arPackVacuum[14];
TransferVacuum5 REF=arPackVacuum[15];
TransferVacuum6 REF=arPackVacuum[16];
TransferVacuum7 REF=arPackVacuum[17];

Check1Cylinder REF= arPackCylinder[41];
Check1Sensor1 REF= arPackSensor[41];
Check1Sensor2 REF= arPackSensor[42];
Check1Sensor3 REF= arPackSensor[43];
Check1Sensor4 REF= arPackSensor[44];
Check1Sensor5 REF= arPackSensor[45];
Check1Sensor6 REF= arPackSensor[46];
Check1Sensor7 REF= arPackSensor[47];

MainRoution();
SR999_Faulthandler();

glb_bUnit01BoxEmpty:= NOT glb_Un01Box.Box[0].Valid 
AND NOT glb_Un01Box.Box[0].Valid AND NOT glb_Un01Box.Box[1].Valid AND NOT glb_Un01Box.Box[2].Valid
AND NOT glb_Un01Box.Box[3].Valid AND NOT glb_Un01Box.Box[4].Valid AND NOT glb_Un01Box.Box[5].Valid
AND NOT glb_Un01Box.Box[6].Valid AND NOT glb_Un01Box.Box[7].Valid AND NOT glb_Un01Box.Box[8].Valid 
AND NOT glb_Un01Box.Box[9].Valid AND NOT glb_Un01Box.Box[10].Valid AND NOT glb_Un01Box.Box[11].Valid
AND NOT glb_Un01Box.Box[12].Valid AND NOT glb_Un01Box.Box[13].Valid AND NOT glb_BoxTransferBuffer.Valid ;

glb_bUnit01BoxNotReady:= NOT glb_Un01Box.Box[HMI_TransferNo-1].Valid 
AND NOT glb_Un01Box.Box[HMI_TransferNo].Valid  AND NOT glb_BoxTransferBuffer.Valid ;

ACTION CM01_Pull:
CASE PullSeq.Now OF
	0:	 
       IF Ref_MachineStateModel.Sts_Execute  THEN
		  PullSeq(ExeCute:= TRUE, Next:= 110); 
	   END_IF	
	   IF Ref_MachineStateModel.Sts_Stopping  THEN
		  PullSeq(ExeCute:= TRUE, Next:= Seq_StoppingDone);  
	   END_IF
	   
	110: 
        PullCylinder1.i.ActiveIn:=TRUE;		PullCylinder1.i.ActiveOut:=FALSE;
        PullCylinder2.i.ActiveIn:=TRUE;		PullCylinder2.i.ActiveOut:=FALSE;
        PullCylinder3.i.ActiveIn:=TRUE;		PullCylinder3.i.ActiveOut:=FALSE;
        PullCylinder4.i.ActiveIn:=TRUE;		PullCylinder4.i.ActiveOut:=FALSE;
        PullCylinder5.i.ActiveIn:=TRUE;		PullCylinder5.i.ActiveOut:=FALSE;
        PullCylinder6.i.ActiveIn:=TRUE;		PullCylinder6.i.ActiveOut:=FALSE;
        PullCylinder7.i.ActiveIn:=TRUE;		PullCylinder7.i.ActiveOut:=FALSE;
		
		IF PullCylinder1.i.InSensor
		AND PullCylinder2.i.InSensor AND PullCylinder3.i.InSensor
		AND PullCylinder4.i.InSensor AND PullCylinder5.i.InSensor
		AND PullCylinder6.i.InSensor AND PullCylinder7.i.InSensor 
		AND NOT PullCylinder1.o.Error AND NOT PullCylinder2.o.Error AND NOT PullCylinder3.o.Error
		AND NOT PullCylinder4.o.Error AND NOT PullCylinder5.o.Error AND NOT PullCylinder6.o.Error
		AND NOT PullCylinder7.o.Error THEN
			PullSeq(ExeCute:= TRUE, Next:= 120);  
		END_IF	
	
	120:
	   IF InfeedSensor1.o.Value AND InfeedSensor2.o.Value AND InfeedSensor3.o.Value AND InfeedSensor4.o.Value AND
		  InfeedSensor5.o.Value AND InfeedSensor6.o.Value AND InfeedSensor7.o.Value THEN
		    PullSeq(ExeCute:= TRUE, Next:= 130);  
		  ELSE IF InfeedSensor8.o.Value AND InfeedSensor9.o.Value AND InfeedSensor10.o.Value AND InfeedSensor11.o.Value AND
		       InfeedSensor12.o.Value AND InfeedSensor13.o.Value AND InfeedSensor14.o.Value THEN
               PullSeq(ExeCute:= TRUE, Next:= 140);  
		  END_IF
	   END_IF
	   
	130:
	   InfeedCylinder.i.ActiveIn:=TRUE;
	   InfeedCylinder.i.ActiveOut:=FALSE;
	   IF InfeedCylinder.i.InSensor AND NOT InfeedCylinder.o.Error THEN
		  PullSeq(ExeCute:= TRUE, Next:= 150);  
	   END_IF   
	   
	140:
	   InfeedCylinder.i.ActiveIn:=FALSE;
	   InfeedCylinder.i.ActiveOut:=TRUE;
	   IF InfeedCylinder.i.OutSensor AND NOT InfeedCylinder.o.Error THEN
		  PullSeq(ExeCute:= TRUE, Next:= 150);  
	   END_IF

	150://计算拉盒数量
	  
		IF NOT bBeltMove AND ref_belt.o.StandStill THEN
			IF (glb_lrBoxTargetCnt<>0) THEN
				PullSeq(ExeCute:= TRUE,Hold:=FALSE, Next:= 160);  
			ELSE IF (glb_lrBoxTargetCnt=0) AND(ref_diTransferFlag<>0) THEN
					 PullSeq(ExeCute:= TRUE,Hold:=FALSE, Next:= 300);  
				 END_IF
			END_IF
		END_IF

		IF Ref_MachineStateModel.Sts_Stopping  THEN
			PullSeq(ExeCute:= TRUE,Hold:=FALSE, Next:= Seq_StoppingDone);  
		END_IF   	   
	   
	   
    160:
        PullCylinder1.i.ActiveIn:=FALSE;		PullCylinder1.i.ActiveOut:=TRUE;
        PullCylinder2.i.ActiveIn:=FALSE;		PullCylinder2.i.ActiveOut:=TRUE;
        PullCylinder3.i.ActiveIn:=FALSE;		PullCylinder3.i.ActiveOut:=TRUE;
        PullCylinder4.i.ActiveIn:=FALSE;		PullCylinder4.i.ActiveOut:=TRUE;
        PullCylinder5.i.ActiveIn:=FALSE;		PullCylinder5.i.ActiveOut:=TRUE;
        PullCylinder6.i.ActiveIn:=FALSE;		PullCylinder6.i.ActiveOut:=TRUE;
        PullCylinder7.i.ActiveIn:=FALSE;		PullCylinder7.i.ActiveOut:=TRUE;
	   
		IF PullCylinder1.i.OutSensor
		AND PullCylinder2.i.OutSensor AND PullCylinder3.i.OutSensor
		AND PullCylinder4.i.OutSensor AND PullCylinder5.i.OutSensor
		AND PullCylinder6.i.OutSensor AND PullCylinder7.i.OutSensor
		AND NOT PullCylinder1.o.Error AND NOT PullCylinder2.o.Error AND NOT PullCylinder3.o.Error
		AND NOT PullCylinder4.o.Error AND NOT PullCylinder5.o.Error AND NOT PullCylinder6.o.Error
		AND NOT PullCylinder7.o.Error THEN
			    PullSeq(ExeCute:= TRUE, Next:= 161); 
		END_IF	
		
	161:
		tonPullSeq(IN:=TRUE , PT:=T#200MS , Q=> , ET=> );
		IF tonPullSeq.Q THEN
			tonPullSeq(IN:=FALSE , PT:=T#200MS , Q=> , ET=> );
			PullSeq(ExeCute:= TRUE, Next:= 162);  
		END_IF
    162:
        //检查真空达到	
		PullVacuum1.i.ActiveIN:=TRUE;
		PullVacuum2.i.ActiveIN:=TRUE;
		PullVacuum3.i.ActiveIN:=TRUE;
		PullVacuum4.i.ActiveIN:=TRUE;
		PullVacuum5.i.ActiveIN:=TRUE;
		PullVacuum6.i.ActiveIN:=TRUE;
		PullVacuum7.i.ActiveIN:=TRUE;	
		IF PullVacuum1.i.Sensor AND PullVacuum2.i.Sensor AND PullVacuum3.i.Sensor AND 
		   PullVacuum4.i.Sensor AND PullVacuum5.i.Sensor AND PullVacuum6.i.Sensor AND PullVacuum7.i.Sensor		
        AND NOT PullVacuum1.o.Error AND NOT PullVacuum2.o.Error AND NOT PullVacuum3.o.Error 
		AND NOT PullVacuum4.o.Error AND NOT PullVacuum5.o.Error AND NOT PullVacuum6.o.Error 
		AND NOT PullVacuum7.o.Error  THEN
		    PullSeq(ExeCute:= TRUE, Next:= 170); 
		END_IF			
 
    170:  
		tonPullSeq(IN:=TRUE , PT:=T#1S , Q=> , ET=> );
		IF tonPullSeq.Q THEN
			tonPullSeq(IN:=FALSE , PT:=T#1S , Q=> , ET=> );
			PullSeq(ExeCute:= TRUE, Next:= 180);  
		END_IF
	   
	180:   
        PullCylinder1.i.ActiveIn:=TRUE;		PullCylinder1.i.ActiveOut:=FALSE;
        PullCylinder2.i.ActiveIn:=TRUE;		PullCylinder2.i.ActiveOut:=FALSE;
        PullCylinder3.i.ActiveIn:=TRUE;		PullCylinder3.i.ActiveOut:=FALSE;
        PullCylinder4.i.ActiveIn:=TRUE;		PullCylinder4.i.ActiveOut:=FALSE;
        PullCylinder5.i.ActiveIn:=TRUE;		PullCylinder5.i.ActiveOut:=FALSE;
        PullCylinder6.i.ActiveIn:=TRUE;		PullCylinder6.i.ActiveOut:=FALSE;
        PullCylinder7.i.ActiveIn:=TRUE;		PullCylinder7.i.ActiveOut:=FALSE;
		
		IF PullCylinder1.i.InSensor
		AND PullCylinder2.i.InSensor AND PullCylinder3.i.InSensor
		AND PullCylinder4.i.InSensor AND PullCylinder5.i.InSensor
		AND PullCylinder6.i.InSensor AND PullCylinder7.i.InSensor 
		AND NOT PullCylinder1.o.Error AND NOT PullCylinder2.o.Error AND NOT PullCylinder3.o.Error
		AND NOT PullCylinder4.o.Error AND NOT PullCylinder5.o.Error AND NOT PullCylinder6.o.Error
		AND NOT PullCylinder7.o.Error THEN
			PullSeq(ExeCute:= TRUE, Next:= 181);  
		END_IF	
		
	181://确保真空未破坏	
		PullVacuum1.i.ActiveIN:=TRUE;
		PullVacuum2.i.ActiveIN:=TRUE;
		PullVacuum3.i.ActiveIN:=TRUE;
		PullVacuum4.i.ActiveIN:=TRUE;
		PullVacuum5.i.ActiveIN:=TRUE;
		PullVacuum6.i.ActiveIN:=TRUE;
		PullVacuum7.i.ActiveIN:=TRUE;	
		IF PullVacuum1.i.Sensor AND PullVacuum2.i.Sensor AND PullVacuum3.i.Sensor AND 
		   PullVacuum4.i.Sensor AND PullVacuum5.i.Sensor AND PullVacuum6.i.Sensor AND PullVacuum7.i.Sensor		
		AND NOT PullVacuum1.o.Error AND NOT PullVacuum2.o.Error AND NOT PullVacuum3.o.Error 
		AND NOT PullVacuum4.o.Error AND NOT PullVacuum5.o.Error AND NOT PullVacuum6.o.Error 
		AND NOT PullVacuum7.o.Error  THEN
			PullSeq(ExeCute:= TRUE, Next:= 190); 
		END_IF		
		
	190:  
		PullVacuum1.i.ActiveIN:=FALSE;
		PullVacuum2.i.ActiveIN:=FALSE;
		PullVacuum3.i.ActiveIN:=FALSE;
		PullVacuum4.i.ActiveIN:=FALSE;
		PullVacuum5.i.ActiveIN:=FALSE;
		PullVacuum6.i.ActiveIN:=FALSE;
		PullVacuum7.i.ActiveIN:=FALSE;
		PullSeq(ExeCute:= TRUE, Next:= 200);  
   
	200:	
		   tonPullSeq(IN:=TRUE , PT:=T#1S , Q=> , ET=> );
		   IF tonPullSeq.Q THEN
			  tonPullSeq(IN:=FALSE , PT:=T#1S , Q=> , ET=> );
			  PullSeq(ExeCute:= TRUE, Next:= 210);  
		   END_IF
		   
	210:
	        glb_lrBoxTargetCnt:=glb_lrBoxTargetCnt-1;
			
	        glb_Un01Box.Box[0].Valid:=TRUE;
			glb_Un01Box.Box[0].Drop:=TRUE;
			glb_Un01Box.Box[0].Cut:=TRUE;
			glb_Un01Box.Box[0].Seal1:=TRUE;
			glb_Un01Box.Box[0].Seal2:=TRUE;			
			glb_Un01Box.Box[0].Transfer:=TRUE;
			glb_Un01Box.Box[0].Check1:=TRUE;
			glb_Un01Box.Box[0].Reject:=TRUE;
			glb_Un01Box.Box[0].PrintData:='END';
			glb_Un01Box.Box[0].amount:=0;
	        bBeltMove:=TRUE;

			ref_diDropFlag.0 :=TRUE;	
			ref_diCutFlag.0 :=TRUE;				
			ref_diSealFlag.0 :=TRUE;	
			ref_diTransferFlag.0 :=TRUE;
			PullSeq(ExeCute:= TRUE,Hold:=FALSE, Next:= 300);  
				
	300:   
			tonPullSeq(IN:=TRUE , PT:=T#1S , Q=> , ET=> );
			IF tonPullSeq.Q THEN
				tonPullSeq(IN:=FALSE , PT:=T#1S , Q=> , ET=> );
				bBeltMove:=TRUE;
				PullSeq(ExeCute:= TRUE,Hold:=FALSE, Next:= 110);  
			END_IF

			
	Seq_StoppingDone:   
	     IF  NOT Ref_MachineStateModel.Sts_Stopping THEN
			 PullSeq(ExeCute:= TRUE, Next:= 0);
		 END_IF	
		 
END_CASE
PullSeq.Hold := Ref_MachineStateModel.Sts_Held;
END_ACTION

ACTION CM02_Drop:
CASE DropSeq.Now OF
	0:	
		IF Ref_MachineStateModel.Sts_Execute  THEN
		   DropSeq(ExeCute:= TRUE, Next:=110); 
		END_IF	
		
		IF Ref_MachineStateModel.Sts_Stopping  THEN
		   DropSeq(ExeCute:= TRUE, Next:= Seq_StoppingDone);    
		END_IF	

	110:
		DropCylinderUP.i.ActiveIn:=TRUE;
		DropCylinderUP.i.ActiveOut:=FALSE;
		DropCylinderDown.i.ActiveIn:=TRUE;
		DropCylinderDown.i.ActiveOut:=FALSE;	
		IF DropCylinderUP.i.InSensor AND  DropCylinderDown.i.InSensor AND 
		NOT DropCylinderUP.o.Error AND NOT DropCylinderDown.o.Error  THEN
			DropSeq(ExeCute:= TRUE, Next:=120);  
		END_IF
	   
	120://等待药品到达     
		IF ref_diDropFlag.2 AND glb_BinBelt4_5.bin[8].arDrop[8] THEN
		   DropSeq(ExeCute:= TRUE,Hold:=FALSE, Next:=121); 
		END_IF
		
		IF Ref_MachineStateModel.Sts_Stopping  THEN
		   DropSeq(ExeCute:= TRUE, Next:= Seq_StoppingDone); 
		END_IF	
		
	121:
	    //判断产品是否需要剔除
	    IF ref_BinList.Bin[49].bReject OR ref_BinList.Bin[48].bReject OR ref_BinList.Bin[47].bReject 
		OR ref_BinList.Bin[46].bReject OR ref_BinList.Bin[45].bReject OR ref_BinList.Bin[44].bReject 
        OR ref_BinList.Bin[43].bReject THEN
		   glb_Un01Box.Box[2].Valid:=FALSE;
		   glb_Un01Box.Box[2].Transfer:=FALSE;
		END_IF
        DropSeq(ExeCute:= TRUE,Hold:=FALSE, Next:=130);
  
	130:   
		DropCylinderUP.i.ActiveIn:=FALSE;
		DropCylinderUP.i.ActiveOut:=TRUE;
		DropCylinderDown.i.ActiveIn:=FALSE;
		DropCylinderDown.i.ActiveOut:=TRUE;	
		IF DropCylinderUP.i.OutSensor AND  DropCylinderDown.i.OutSensor AND 
		NOT DropCylinderUP.o.Error AND NOT DropCylinderDown.o.Error  THEN
			DropSeq(ExeCute:= TRUE, Next:= 131);  
		END_IF

	131:   
		tonDropSeq(IN:=TRUE , PT:=T#1500MS , Q=> , ET=> );
		IF tonDropSeq.Q THEN
		   tonDropSeq(IN:=FALSE , PT:=T#1500MS , Q=> , ET=> );
		   DropSeq(ExeCute:= TRUE, Next:= 140); 
		END_IF	

	140:
		DropCylinderUP.i.ActiveIn:=TRUE;
		DropCylinderUP.i.ActiveOut:=FALSE;
		IF DropCylinderUp.i.InSensor AND NOT  DropCylinderUP.o.Error THEN
		   DropSeq(ExeCute:= TRUE, Next:= 141);     
		END_IF	
			
	141:
        IF 	glb_BinBelt4_5.bin[9].arDrop[8] THEN 
			glb_Un01Box.Box[HMI_DropNo].PrintData:=glb_BinBelt4_5.bin[9].Name;
			glb_Un01Box.Box[HMI_DropNo].amount:=glb_BinBelt4_5.bin[9].Amount;
			(*
			glb_Un01Box.Box[HMI_DropNo].Reject:=glb_BinBelt4_5.bin[9].bReject
            OR glb_BinBelt4_5.bin[8].bReject OR glb_BinBelt4_5.bin[7].bReject
            OR glb_BinBelt4_5.bin[6].bReject OR glb_BinBelt4_5.bin[5].bReject
            OR glb_BinBelt4_5.bin[4].bReject OR glb_BinBelt4_5.bin[3].bReject;
			*)
			glb_BinBelt4_5.bin[9].arDrop[8]:=FALSE;
			glb_BinBelt4_5.bin[8].arDrop[8]:=FALSE;
			glb_BinBelt4_5.bin[7].arDrop[8]:=FALSE;
			glb_BinBelt4_5.bin[6].arDrop[8]:=FALSE;
			glb_BinBelt4_5.bin[5].arDrop[8]:=FALSE;
			glb_BinBelt4_5.bin[4].arDrop[8]:=FALSE;
			glb_BinBelt4_5.bin[3].arDrop[8]:=FALSE;
						
        ELSE IF glb_BinBelt4_5.bin[8].arDrop[8] THEN
			    glb_Un01Box.Box[HMI_DropNo].PrintData:=glb_BinBelt4_5.bin[8].Name;
				glb_Un01Box.Box[HMI_DropNo].amount:=glb_BinBelt4_5.bin[8].Amount;
				(*
				glb_Un01Box.Box[HMI_DropNo].Reject:=glb_BinBelt4_5.bin[8].bReject
				OR glb_BinBelt4_5.bin[2].bReject OR glb_BinBelt4_5.bin[7].bReject
				OR glb_BinBelt4_5.bin[6].bReject OR glb_BinBelt4_5.bin[5].bReject
				OR glb_BinBelt4_5.bin[4].bReject OR glb_BinBelt4_5.bin[3].bReject;	
                *)
			
				glb_BinBelt4_5.bin[8].arDrop[8]:=FALSE;
				glb_BinBelt4_5.bin[7].arDrop[8]:=FALSE;
				glb_BinBelt4_5.bin[6].arDrop[8]:=FALSE;
				glb_BinBelt4_5.bin[5].arDrop[8]:=FALSE;
				glb_BinBelt4_5.bin[4].arDrop[8]:=FALSE;
				glb_BinBelt4_5.bin[3].arDrop[8]:=FALSE;
			 	glb_BinBelt4_5.bin[2].arDrop[8]:=FALSE;	
		
		     END_IF
		END_IF
		
		ref_Work_Recipe.OutQuantity:=ref_Work_Recipe.OutQuantity+7;
		DropSeq(ExeCute:= TRUE,Hold:=FALSE, Next:= 142); 
			
    142:  
		tonDropSeq(IN:=TRUE , PT:=T#2000MS , Q=> , ET=> );   
		IF tonDropSeq.Q THEN
			tonDropSeq(IN:=FALSE , PT:=T#2000MS , Q=> , ET=> );
			DropSeq(ExeCute:= TRUE, Next:= 150); 
		END_IF	
	150:
		DropCylinderDown.i.ActiveIn:=TRUE;
		DropCylinderDown.i.ActiveOut:=FALSE;	 
		IF DropCylinderDown.i.InSensor AND NOT DropCylinderDown.o.Error THEN
			DropSeq(ExeCute:= TRUE, Next:= 160);   
		END_IF	
			
	160:
		ref_diDropFlag.2:=0;
		ref_diGoodFlag.2:=1;
		DropSeq(ExeCute:= TRUE,Hold:=FALSE, Next:= 110); 		
			
	Seq_StoppingDone:
			 IF  NOT Ref_MachineStateModel.Sts_Stopping THEN
				 DropSeq(ExeCute:= TRUE, Next:= 0); 
			 END_IF			
END_CASE
DropSeq.Hold := Ref_MachineStateModel.Sts_Held;
END_ACTION

ACTION CM03_Cut:
CASE CutSeq.Now OF	
	0:
	   IF Ref_MachineStateModel.Sts_Execute  THEN
		  CutSeq(Execute:= TRUE, Next:= 110);  
          //CutSeq(Execute:= TRUE, Next:= 0);   
		  //ref_diCutFlag.8 :=FALSE;
	   END_IF	
	
	   IF Ref_MachineStateModel.Sts_Stopping THEN
		  CutSeq(Execute:= TRUE, Next:= Seq_StoppingDone);     
	   END_IF	
	
	110:
		tonCutSeq(IN:=TRUE , PT:=T#1S , Q=> , ET=> );
		IF tonCutSeq.Q THEN
			tonCutSeq(IN:=FALSE , PT:=T#1S , Q=> , ET=> );
			CutSeq(Execute:= TRUE,Hold:=FALSE, Next:= 111); 
		END_IF	

    111:
		lrEncoderPosOld:=ref_Encoder.NcToPlc.ActPos;
		ref_WindMotor.Backward:=TRUE;
		ref_Puller.i.Enable:=TRUE;
		IF ref_Puller.o.PowerOn THEN
		   CutSeq(Execute:= TRUE, Next:= 120);  
		END_IF  
				
	120:
		tonCutSeq(IN:=TRUE , PT:=T#10S , Q=> , ET=> );		
		ref_Puller.i.JogP:=TRUE;
		IF ref_Encoder.NcToPlc.ActPos-lrEncoderPosOld > ref_Puller.i.Pos-6 THEN
			ref_Puller.i.JogP:=FALSE; 
			tonCutSeq(IN:=FALSE , PT:=T#10S , Q=> , ET=> );
            CutSeq(Execute:= TRUE,Hold:=FALSE, Next:= 130); 	
			ELSE IF tonCutSeq.Q THEN
			        glb_MembraneAlarm:=TRUE;
					ref_Puller.i.JogP:=FALSE; 
					tonCutSeq(IN:=FALSE , PT:=T#10S , Q=> , ET=> );
					CutSeq(Execute:= TRUE,Hold:=FALSE, Next:= 121); 				  
			     END_IF	
		END_IF
    121:
		IF NOT glb_MembraneAlarm THEN
			CutSeq(Execute:= TRUE,Hold:=FALSE, Next:= 110); 
		END_IF
		IF Ref_MachineStateModel.Sts_Stopping THEN
			CutSeq(Execute:= TRUE, Next:= Seq_StoppingDone);     
		END_IF			
	130:
		tonCutSeq(IN:=TRUE , PT:=T#1S , Q=> , ET=> );
		IF tonCutSeq.Q THEN
			tonCutSeq(IN:=FALSE , PT:=T#1S , Q=> , ET=> );
			CutSeq(Execute:= TRUE,Hold:=FALSE, Next:= 140); 
		END_IF	
		
	140:		
		IF ref_diCutFlag.7 THEN
		   CutSeq(Execute:= TRUE, Next:= 141); 
		END_IF
		IF Ref_MachineStateModel.Sts_Stopping THEN
		   CutSeq(Execute:= TRUE, Next:= Seq_Stopping);  
		END_IF	
	141:
        IF glb_Un01Box.Box[HMI_Seal1No].Seal1 THEN//IF ref_diSealFlag.10 THEN
           CutSeq(Execute:= TRUE, Next:= 142);
        ELSE 
           CutSeq(Execute:= TRUE, Next:= 150); 
        END_IF
		
    142:     
         IF SealCylinderDown.i.OutSensor OR glb_Un01Box.Box[HMI_Seal1No].Seal1 THEN
	     //IF SealCylinderDown.i.OutSensor OR NOT ref_diSealFlag.10 THEN
			CutSeq(Execute:= TRUE, Next:= 150);   
		 END_IF
		 IF Ref_MachineStateModel.Sts_Stopping THEN
		    CutSeq(Execute:= TRUE, Next:= Seq_Stopping);  
		 END_IF	 
		 
	150: 
		CutCylinderDown.i.ActiveIn:=FALSE;
		CutCylinderDown.i.ActiveOut:=TRUE;
		IF  CutCylinderDown.i.OutSensor AND NOT CutCylinderDown.o.Error  THEN
		 	CutSeq(Execute:= TRUE, Next:= 160); 
		END_IF	  
	  
	160:
		CutCylinderUp.i.ActiveIn:=FALSE;
		CutCylinderUp.i.ActiveOut:=TRUE;
		IF  CutCylinderUp.i.OutSensor AND NOT CutCylinderUp.o.Error  THEN
		 	CutSeq(Execute:= TRUE, Next:= 161); 
		END_IF		
		
	161:	
		tonCutSeq(IN:=TRUE , PT:=T#1S , Q=> , ET=> );
		IF tonCutSeq.Q THEN
			tonCutSeq(IN:=FALSE , PT:=T#1S , Q=> , ET=> );
			CutSeq(Execute:= TRUE,Hold:=FALSE, Next:= 170); 
		END_IF	

	170:
		CutCylinderUp.i.ActiveIn:=TRUE;
		CutCylinderUp.i.ActiveOut:=FALSE;
		IF CutCylinderUp.i.InSensor AND NOT CutCylinderUp.o.Error THEN
		    CutSeq(Execute:= TRUE, Next:= 171); 
		END_IF		    
 
    171: 
		CutCylinderDown.i.ActiveIn:=TRUE;
		CutCylinderDown.i.ActiveOut:=FALSE;
		IF CutCylinderDown.i.InSensor AND NOT CutCylinderDown.o.Error  THEN
		    CutSeq(Execute:= TRUE, Next:= 180); 
		END_IF
	
	
    180:
		  ref_diCutFlag.7 :=FALSE;
		  CutSeq(Execute:= TRUE,Hold:=FALSE, Next:= 110); 
	 
	 
	 
    Seq_Stopping:

		ref_Puller.i.jogP:=FALSE;       
        IF NOT ref_Puller.o.StandStill THEN
		   ref_Puller.i.stop:=TRUE;       
        ELSE
		   ref_Puller.i.Stop:=FALSE;
	       CutSeq(Execute:= TRUE,Hold:=FALSE, Next:= Seq_StoppingDone);
		END_IF   
	 
	 
	Seq_StoppingDone:
	
		 ref_Puller.i.Enable:=FALSE;
		 ref_WindMotor.Forward:=FALSE;
		 ref_WindMotor.Backward:=FALSE;		 
		 ref_Puller.i.JogP:=FALSE;
		 IF  NOT Ref_MachineStateModel.Sts_Stopping THEN
			 CutSeq(Execute:= TRUE,Hold:=FALSE, Next:= 0); 
		 END_IF		 
 
END_CASE
CutSeq.Hold := Ref_MachineStateModel.Sts_Held;
END_ACTION

ACTION CM04_Transfer:
TransferSeq(ExeCute:= TRUE, Next:= , Last=> , Now=> );
CASE TransferSeq.Now OF
	0:	
	   IF Ref_MachineStateModel.Sts_Execute  THEN
		  TransferSeq(ExeCute:= TRUE, Next:= 110);  
	   END_IF	
	
	   IF Ref_MachineStateModel.Sts_Stopping  THEN
		  TransferSeq(ExeCute:= TRUE, Next:= Seq_StoppingDone);     
	   END_IF	
	   
	110:
	   TransferCyliderVert.i.ActiveIn:=TRUE;
	   TransferCyliderVert.i.ActiveOut:=FALSE;	   
	   IF TransferCyliderVert.i.InSensor AND NOT TransferCyliderVert.o.Error  THEN
		  TransferSeq(ExeCute:= TRUE, Next:= 120);  
	   END_IF
	   
	120:

	   TransferCyliderRota.i.ActiveIn:=TRUE;
	   TransferCyliderRota.i.ActiveOut:=FALSE;	   
	   IF  TransferCyliderRota.i.InSensor AND NOT TransferCyliderRota.o.Error  THEN
		   TransferSeq(ExeCute:= TRUE, Next:= 130);  
	   END_IF   
	   
	130:
	   TransferCyliderHori.i.ActiveIn:=FALSE;
	   TransferCyliderHori.i.ActiveOut:=TRUE;	   
	   IF TransferCyliderHori.i.OutSensor AND NOT TransferCyliderHori.o.Error THEN
		  TransferSeq(ExeCute:= TRUE, Next:= 140);  
	   END_IF   
	
	140://等待产品到达
	   //IF ref_diTransferFlag.13 THEN
	   IF glb_Un01Box.Box[HMI_TransferNo].Transfer THEN
		  TransferSeq(ExeCute:= TRUE, Next:= 150);  
	   END_IF 
	   IF Ref_MachineStateModel.Sts_Stopping  THEN
		  TransferSeq(ExeCute:= TRUE, Next:= Seq_StoppingDone);    
	   END_IF
		
	150:
	   
	   TransferCyliderVert.i.ActiveIn:=FALSE;
	   TransferCyliderVert.i.ActiveOut:=TRUE;	
	   IF TransferCyliderVert.i.OutSensor AND NOT TransferCyliderVert.o.Error THEN
		  TransferSeq(ExeCute:= TRUE, Next:= 160);  
	   END_IF
	   
	160: //开真空
		TransferVacuum1.i.ActiveIN:=TRUE;
		TransferVacuum2.i.ActiveIN:=TRUE;
		TransferVacuum3.i.ActiveIN:=TRUE;
		TransferVacuum4.i.ActiveIN:=TRUE;
		TransferVacuum5.i.ActiveIN:=TRUE;
		TransferVacuum6.i.ActiveIN:=TRUE;
		TransferVacuum7.i.ActiveIN:=TRUE;	
		
		tonTransferSeq(IN:=TRUE , PT:=T#2S , Q=> , ET=> );
		IF tonTransferSeq.Q THEN
			tonTransferSeq(IN:=FALSE , PT:=T#2S , Q=> , ET=> );
			TransferSeq(ExeCute:= TRUE,Hold:=FALSE, Next:= 170);  
		END_IF	
			
    170:
	   TransferCyliderVert.i.ActiveIn:=TRUE;
	   TransferCyliderVert.i.ActiveOut:=FALSE;
	   IF TransferCyliderVert.i.InSensor AND NOT TransferCyliderVert.o.Error THEN
		  TransferSeq(ExeCute:= TRUE, Next:= 171);  
	   END_IF	
	   
	171://检查真空
	    IF TransferVacuum1.i.Sensor AND TransferVacuum2.i.Sensor AND TransferVacuum3.i.Sensor AND 
		TransferVacuum4.i.Sensor AND  TransferVacuum5.i.Sensor AND  TransferVacuum6.i.Sensor AND
		TransferVacuum7.i.Sensor AND NOT TransferVacuum1.o.Error AND NOT TransferVacuum2.o.Error 
		AND NOT TransferVacuum3.o.Error AND NOT TransferVacuum4.o.Error AND NOT TransferVacuum5.o.Error
		AND NOT TransferVacuum6.o.Error AND NOT TransferVacuum7.o.Error THEN
		TransferSeq(ExeCute:= TRUE, Next:= 172);
		END_IF
	172:
		tonTransferSeq(IN:=TRUE , PT:=T#1S , Q=> , ET=> );
		IF tonTransferSeq.Q THEN
			tonTransferSeq(IN:=FALSE , PT:=T#1S , Q=> , ET=> );
			TransferSeq(ExeCute:= TRUE,Hold:=FALSE, Next:= 173);  
		END_IF		
		
	173:
		ref_diTransferFlag.13 :=0;
		ref_diGoodFlag.13 :=0;
		ref_diNoGoodFlag.13 :=0;
		glb_Un01Box.Box[HMI_TransferNo].Transfer:=FALSE;
		glb_BoxTransferBuffer:=glb_Un01Box.Box[HMI_TransferNo];//纸盒数据复制到缓冲区
		TransferSeq(ExeCute:= TRUE,Hold:=FALSE, Next:= 174);
		
    174:
		MEMSET(destAddr:= ADR(glb_Un01Box.Box[HMI_TransferNo]), fillByte:= 0, n:= SIZEOF(glb_Un01Box.Box[11]));		
		TransferSeq(ExeCute:= TRUE,Hold:=FALSE, Next:= 180);
  		  
	180:   
		TransferCyliderHori.i.ActiveIn:=TRUE;
		TransferCyliderHori.i.ActiveOut:=FALSE;
		IF TransferCyliderHori.i.InSensor AND NOT TransferCyliderHori.o.Error  THEN
		   TransferSeq(ExeCute:= TRUE, Next:= 181);  
		END_IF	
		
    181:
		tonTransferSeq(IN:=TRUE , PT:=T#1.5S , Q=> , ET=> );
		IF tonTransferSeq.Q THEN
			tonTransferSeq(IN:=FALSE , PT:=T#1.5S , Q=> , ET=> );
			TransferSeq(ExeCute:= TRUE, Next:= 190);  
		END_IF			
		
		
    190:
		IF ref_bTransferPut OR HMI_SkipTransferPut THEN
		   TransferSeq(ExeCute:= TRUE, Next:= 200);  
		END_IF
	
	200:
		TransferCyliderVert.i.ActiveIn:=FALSE;
		TransferCyliderVert.i.ActiveOut:=TRUE;
		IF TransferCyliderVert.i.OutSensor AND NOT TransferCyliderVert.o.Error  THEN
		   TransferSeq(ExeCute:= TRUE, Next:= 210);  
		END_IF	
	 
		
	210:  
	   	TransferVacuum1.i.ActiveIN:=FALSE;
		TransferVacuum2.i.ActiveIN:=FALSE;
		TransferVacuum3.i.ActiveIN:=FALSE;
		TransferVacuum4.i.ActiveIN:=FALSE;
		TransferVacuum5.i.ActiveIN:=FALSE;
		TransferVacuum6.i.ActiveIN:=FALSE;
		TransferVacuum7.i.ActiveIN:=FALSE;
		tonTransferSeq(IN:=TRUE , PT:=T#2S , Q=> , ET=> );
		IF tonTransferSeq.Q THEN
			tonTransferSeq(IN:=FALSE , PT:=T#2S , Q=> , ET=> );
			TransferSeq(ExeCute:= TRUE, Next:= 220);  
		END_IF	
		
	 220:
		TransferCyliderVert.i.ActiveIn:=TRUE;
		TransferCyliderVert.i.ActiveOut:=FALSE;	   
		IF TransferCyliderVert.i.InSensor AND NOT TransferCyliderVert.o.Error  THEN
		   TransferSeq(ExeCute:= TRUE, Next:= 221);  
		END_IF
	
     221:
		tonTransferSeq(IN:=TRUE , PT:=T#1.5S , Q=> , ET=> );
		IF tonTransferSeq.Q THEN
			tonTransferSeq(IN:=FALSE , PT:=T#1.5S , Q=> , ET=> );
			TransferSeq(ExeCute:= TRUE, Next:= 230);  
		END_IF	
		
	 230:
	    glb_Un02Box.Box[0]:=glb_BoxTransferBuffer;//缓冲区纸盒传递到皮带7
		glb_Un02Box.Box[0].PrintRequest:=TRUE;
	    TransferSeq(ExeCute:= TRUE,Hold:=FALSE, Next:= 240); 	
	 240:	
		MEMSET(destAddr:= ADR(glb_BoxTransferBuffer), fillByte:= 0, n:= SIZEOF(glb_BoxTransferBuffer));
		ref_bTransferPut:=FALSE;
		glb_TransferCnt:=glb_TransferCnt+1;
		TransferSeq(ExeCute:= TRUE,Hold:=FALSE, Next:= 110);   
	
	Seq_StoppingDone:
		 IF  NOT Ref_MachineStateModel.Sts_Stopping THEN
			 TransferSeq(ExeCute:= TRUE, Next:= 0);  
		 END_IF		
END_CASE
TransferSeq.Hold := Ref_MachineStateModel.Sts_Held;
END_ACTION

ACTION CM05_Belt:
CASE BeltSeq.Now  OF	
	0:	
	   IF Ref_MachineStateModel.Sts_Resetting THEN
		  BeltSeq(Execute:= TRUE, Next:= Seq_Resetting);   
	   END_IF
	
	   IF Ref_MachineStateModel.Sts_Execute  THEN
		  BeltSeq(Execute:= TRUE, Next:= 110);     
	   END_IF	
	
	   IF Ref_MachineStateModel.Sts_Stopping  THEN
		  BeltSeq(Execute:= TRUE, Next:= Seq_Stopping);   
	   END_IF
	
	Seq_Resetting:
		IF NOT ref_Belt.o.PowerOn  THEN;
		   ref_Belt.i.Enable:=TRUE;
		END_IF	
		IF NOT ref_Puller.o.PowerOn  THEN;
		   ref_Puller.i.Enable:=TRUE;
		END_IF		
		IF ref_Belt.o.PowerOn AND ref_Puller.o.PowerOn AND HomeValve() THEN
		   BeltSeq(Execute:= TRUE, Next:= 20);   
		END_IF
		IF Ref_MachineStateModel.Sts_Stopping  THEN
		   BeltSeq(Execute:= TRUE, Next:= Seq_Stopping);   
		END_IF	
		
	20:
		IF NOT glb_AllAxisHomed_UN01  THEN
			BeltSeq(Execute:= TRUE, Next:= 21);   
			ELSE
			BeltSeq(Execute:= TRUE, Next:= 30);   	  
		END_IF
		
	21://回零复位
	    glb_lrBoxTargetCnt:=0;
		glb_lrBoxWrkCnt:=0;
        MEMSET(destAddr:= ADR(glb_Un01Box), fillByte:= 0, n:= SIZEOF(glb_Un01Box));  
	    BeltSeq(Execute:= TRUE, Next:= 22);     
	   
	22:
	   tonBeltSeq(IN:=TRUE , PT:=T#1S , Q=> , ET=> );
	   IF tonBeltSeq.Q THEN
		  tonBeltSeq(IN:=FALSE , PT:=T#1S , Q=> , ET=> );
		  ref_Belt.i.HomeMode:=0;//
	      ref_Belt.i.Home:=TRUE;
		  BeltSeq(Execute:= TRUE, Next:= 23);   
	   END_IF
	  
	23:   
	   IF ref_Belt.o.HomeDone THEN
			ref_Belt.i.Home:=FALSE;
			BeltSeq(Execute:= TRUE, Next:= 24);   
	   ELSE IF Ref_MachineStateModel.Sts_Stopping  THEN
		       ref_Belt.i.Home:=FALSE;
               BeltSeq(Execute:= TRUE, Next:= Seq_Stopping);     
	        END_IF
	   END_IF
	   
	24:
	    lrPosCnt:=1;
		bBeltMove:=FALSE;
		ref_Belt.i.Pos:=0;
		ref_diTransferFlag:=0;
        ref_diCutFlag:=0; 		
        ref_diSealFlag:=0; 
	    ref_diDropFlag:=0;
        ref_diPullFlag:=0;
        BeltSeq(Execute:= TRUE, Next:= 25);   
		
	25:
        IF ref_Belt.o.StandStill THEN
		   BeltSeq(Execute:= TRUE, Next:= 30);   
	    END_IF
		
    30:	//生产复位
	    ref_Belt.i.MoveAbs:=TRUE;
	    BeltSeq(Execute:= TRUE, Next:= 31);   	
		
	31:
    	IF  ref_Belt.o.CmdDone THEN
		    ref_Belt.i.MoveAbs:=FALSE;
            BeltSeq(Execute:= TRUE, Next:= Seq_ResettingDone);    	
		END_IF

   
	110:
		   IF NOT glb_Un01Box.Box[HMI_TransferNo].Transfer // ref_diTransferFalg.12
           AND NOT glb_Un01Box.Box[HMI_Seal2No].Seal2 //  ref_diSealFlag.10  
		   AND NOT glb_Un01Box.Box[HMI_Seal1No].Seal1 //  ref_diSealFlag.10 
		   AND NOT ref_diCutFlag.7 
		   AND NOT ref_diDropFlag.2
		   AND NOT glb_Un01Box.Box[HMI_Check1No].Check1
		   AND NOT bRejectActive
		   AND bBeltMove THEN
			  BeltSeq(Execute:= TRUE, Next:= 120);   
		   END_IF
		   IF Ref_MachineStateModel.Sts_Stopping  THEN
			  BeltSeq(Execute:= TRUE, Next:= Seq_Stopping);   
		   END_IF
       
	120: 
		ref_belt.i.Pos:=222.25*LrPosCnt; 
		ref_belt.i.MoveABS:=TRUE;
		BeltSeq(Execute:= TRUE, Next:= 130);
		
	130: 	
        IF ref_belt.o.CmdDone THEN
		   ref_belt.i.MoveABS:=FALSE;	
		   BeltSeq(Execute:= TRUE,Hold:=FALSE, Next:= 140);		
		END_IF
	    
	140: 
	    LrPosCnt:=LrPosCnt+1;
		bRejectActive:=TRUE;
        ref_diDropFlag:=SHL(ref_diDropFlag,1);	
		ref_diCutFlag:=SHL(ref_diSealFlag,1);	
		ref_diSealFlag:=SHL(ref_diSealFlag,1);	
		ref_diTransferFlag:=SHL(ref_diTransferFlag,1);

        ref_diGoodFlag:=SHL(ref_diGoodFlag,1);	
		ref_diNogoodFlag:=SHL(ref_diNogoodFlag,1);	
	
		FOR iBox:= 63 TO 1 BY -1 DO
			glb_Un01Box.Box[iBox]:=glb_Un01Box.Box[iBox-1];
		END_FOR		
     	BeltSeq(Execute:= TRUE,Hold:=FALSE, Next:= 150);
		
    150:    
		glb_Un01Box.Box[0].Valid:=FALSE;
		glb_Un01Box.Box[0].Drop:=FALSE;
		glb_Un01Box.Box[0].Cut:=FALSE;
		glb_Un01Box.Box[0].Seal1:=FALSE;
		glb_Un01Box.Box[0].Seal2:=FALSE;			
		glb_Un01Box.Box[0].Transfer:=FALSE;
		glb_Un01Box.Box[0].Check1:=FALSE;
	    BeltSeq(Execute:= TRUE,Hold:=FALSE, Next:= 160);
		
	160:	
		bBeltMove:=FALSE;		
	    BeltSeq(Execute:= TRUE,Hold:=FALSE, Next:= 110);
	
    Seq_Stopping:
        IF NOT ref_belt.o.StandStill THEN
		   ref_belt.i.stop:=TRUE;       
        ELSE
		   ref_belt.i.Stop:=FALSE;
	       BeltSeq(Execute:= TRUE, Next:= Seq_StoppingDone);
		END_IF   
	
	Seq_ResettingDone:
		IF NOT Ref_MachineStateModel.Sts_Resetting THEN
			BeltSeq(Execute:= TRUE, Next:= 0);
		END_IF	
	
    Seq_stoppingDone:	
	     ref_belt.i.disable:=TRUE;
		 IF  NOT Ref_MachineStateModel.Sts_Stopping THEN
			 BeltSeq(Execute:= TRUE, Next:= 0);
		 END_IF	
		
END_CASE 
BeltSeq.Hold := Ref_MachineStateModel.Sts_Held;
END_ACTION

ACTION CM06_Seal:
bBoxSealView:=
glb_Un01Box.Box[1].Seal1 OR glb_Un01Box.Box[2].Seal1 OR glb_Un01Box.Box[3].Seal1 OR glb_Un01Box.Box[4].Seal1 OR
 glb_Un01Box.Box[5].Seal1 OR glb_Un01Box.Box[6].Seal1 OR glb_Un01Box.Box[7].Seal1 OR glb_Un01Box.Box[8].Seal1 OR
 glb_Un01Box.Box[9].Seal1 OR glb_Un01Box.Box[10].Seal1 ;

CASE SealSeq.Now OF	
	0:
	   IF Ref_MachineStateModel.Sts_Execute  THEN
		  SealSeq(Execute:= TRUE, Next:= 110);  
          //SealSeq(Execute:= TRUE, Next:= 0);   
		  //ref_diSealFlag.11 :=FALSE;
	   END_IF	
	
	   IF Ref_MachineStateModel.Sts_Stopping THEN
		  SealSeq(Execute:= TRUE, Next:= Seq_StoppingDone);     
	   END_IF	
	
	110:   	
		IF glb_Un01Box.Box[HMI_Seal1No].Seal1 THEN//ref_diSealFlag.10 THEN
		   SealSeq(Execute:= TRUE, Next:= 120); 
		END_IF
		IF Ref_MachineStateModel.Sts_Stopping THEN
		   SealSeq(Execute:= TRUE, Next:= Seq_StoppingDone);  
		END_IF	
		
	120: 
		SealCylinderDown.i.ActiveIn:=FALSE;
		SealCylinderDown.i.ActiveOut:=TRUE;
		IF  SealCylinderDown.i.OutSensor AND NOT SealCylinderDown.o.Error  THEN
		 	SealSeq(Execute:= TRUE, Next:= 121); 
		END_IF	  
		
	121:
		tonSealSeq(IN:=TRUE , PT:=T#1S , Q=> , ET=> );
		IF tonSealSeq.Q THEN
			tonSealSeq(IN:=FALSE , PT:=T#1S, Q=> , ET=> );
			SealSeq(Execute:= TRUE,Hold:=FALSE, Next:= 130); 
		END_IF	
 
	130:
		SealCylinderUp.i.ActiveIn:=FALSE;
		SealCylinderUp.i.ActiveOut:=TRUE;
		SealSeq(Execute:= TRUE,Hold:=FALSE, Next:= 140); 
	  
	  	  
	140://封口保压
		tonSealSeq(IN:=TRUE , PT:=DINT_TO_TIME(HMI_SealTime) , Q=> , ET=> );
		IF tonSealSeq.Q THEN
			tonSealSeq(IN:=FALSE , PT:=DINT_TO_TIME(HMI_SealTime) , Q=> , ET=> );
			SealSeq(Execute:= TRUE,Hold:=FALSE, Next:= 150); 
		END_IF	
   
    150: 
	
		SealCylinderUp.i.ActiveIn:=TRUE;
		SealCylinderUp.i.ActiveOut:=FALSE;
		IF SealCylinderUp.i.InSensor 
		AND NOT SealCylinderUp.o.Error THEN
		    SealSeq(Execute:= TRUE, Next:= 151); 
		END_IF		
		
	151:
	    IF HMI_arSealTime[1]<>0 THEN
	       SealSeq(Execute:= TRUE, Next:= 160);		
        ELSE
	       SealSeq(Execute:= TRUE, Next:= 180);		
		END_IF
	

 
	160:
		SealCylinderUp.i.ActiveIn:=FALSE;
		SealCylinderUp.i.ActiveOut:=TRUE;
		SealSeq(Execute:= TRUE,Hold:=FALSE, Next:= 170); 
	  
	  	  
	170://封口保压
		tonSealSeq(IN:=TRUE , PT:=DINT_TO_TIME(HMI_arSealTime[1]) , Q=> , ET=> );
		IF tonSealSeq.Q THEN
			tonSealSeq(IN:=FALSE , PT:=DINT_TO_TIME(HMI_arSealTime[1]) , Q=> , ET=> );
			SealSeq(Execute:= TRUE,Hold:=FALSE, Next:= 180); 
		END_IF	
		
	180:
		SealCylinderUp.i.ActiveIn:=TRUE;
		SealCylinderUp.i.ActiveOut:=FALSE;		
		SealCylinderDown.i.ActiveIn:=TRUE;
		SealCylinderDown.i.ActiveOut:=FALSE;
		IF SealCylinderDown.i.InSensor AND SealCylinderUp.i.InSensor 
		AND NOT SealCylinderDown.o.Error 
		AND NOT SealCylinderUp.o.Error THEN
			SealSeq(Execute:= TRUE, Next:= 190); 
		END_IF
	
  
	190:
		  ref_diSealFlag.10 :=FALSE;
		  glb_Un01Box.Box[HMI_Seal1No].Seal1:=FALSE;
		  SealSeq(Execute:= TRUE,Hold:=FALSE, Next:= 110); 


	 
	Seq_StoppingDone:
		 IF  NOT Ref_MachineStateModel.Sts_Stopping THEN
			 SealSeq(Execute:= TRUE, Next:= 0); 
		 END_IF		 
 
END_CASE
SealSeq.Hold := Ref_MachineStateModel.Sts_Held;
END_ACTION

ACTION CM07_Seal2:
CASE Seal2Seq.Now OF	
	0:
	   IF Ref_MachineStateModel.Sts_Execute  THEN
		  Seal2Seq(Execute:= TRUE, Next:= 110);  
	   END_IF	
	
	   IF Ref_MachineStateModel.Sts_Stopping THEN
		  Seal2Seq(Execute:= TRUE, Next:= Seq_StoppingDone);     
	   END_IF	
	
	110:   	
		IF glb_Un01Box.Box[HMI_Seal2No].Seal2 THEN
		   Seal2Seq(Execute:= TRUE, Next:= 111); 
		END_IF
		IF Ref_MachineStateModel.Sts_Stopping THEN
		   Seal2Seq(Execute:= TRUE, Next:= Seq_StoppingDone);  
		END_IF	
	111:
        IF SealCylinderDown.i.OutSensor OR NOT glb_Un01Box.Box[HMI_Seal1No].Seal1 THEN
		   Seal2Seq(Execute:= TRUE, Next:= 120);
		END_IF
		IF Ref_MachineStateModel.Sts_Stopping THEN
		   Seal2Seq(Execute:= TRUE, Next:= Seq_StoppingDone);  
		END_IF	
		
	120: 
		Seal2CylinderDown.i.ActiveIn:=FALSE;
		Seal2CylinderDown.i.ActiveOut:=TRUE;
		IF  Seal2CylinderDown.i.OutSensor AND NOT Seal2CylinderDown.o.Error  THEN
		 	Seal2Seq(Execute:= TRUE, Next:= 121); 
		END_IF	  
		
	121:
		tonSeal2Seq(IN:=TRUE , PT:=T#1S , Q=> , ET=> );
		IF tonSeal2Seq.Q THEN
			tonSeal2Seq(IN:=FALSE , PT:=T#1S , Q=> , ET=> );
			Seal2Seq(Execute:= TRUE,Hold:=FALSE, Next:= 130); 
		END_IF	
 
	130:
		Seal2CylinderUp.i.ActiveIn:=FALSE;
		Seal2CylinderUp.i.ActiveOut:=TRUE;
		Seal2Seq(Execute:= TRUE,Hold:=FALSE, Next:= 140); 
	  
	  	  
	140://封口保压
		tonSeal2Seq(IN:=TRUE , PT:=DINT_TO_TIME(HMI_SealTime2) , Q=> , ET=> );
		IF tonSeal2Seq.Q THEN
			tonSeal2Seq(IN:=FALSE , PT:=DINT_TO_TIME(HMI_SealTime2) , Q=> , ET=> );
			Seal2Seq(Execute:= TRUE,Hold:=FALSE, Next:= 150); 
		END_IF	
   
    150: 
		Seal2CylinderUp.i.ActiveIn:=TRUE;
		Seal2CylinderUp.i.ActiveOut:=FALSE;
		IF Seal2CylinderUp.i.InSensor 
		AND NOT Seal2CylinderUp.o.Error THEN
		    Seal2Seq(Execute:= TRUE, Next:= 180); 
		END_IF		
	(*	
	160:
		Seal2CylinderUp.i.ActiveIn:=FALSE;
		Seal2CylinderUp.i.ActiveOut:=TRUE;
		Seal2Seq(Execute:= TRUE,Hold:=FALSE, Next:= 170); 
	  
	  	  
	170://封口保压
		tonSeal2Seq(IN:=TRUE , PT:=DINT_TO_TIME(HMI_arSealTime[1]) , Q=> , ET=> );
		IF tonSeal2Seq.Q THEN
			tonSeal2Seq(IN:=FALSE , PT:=DINT_TO_TIME(HMI_arSealTime[1]) , Q=> , ET=> );
			Seal2Seq(Execute:= TRUE,Hold:=FALSE, Next:= 180); 
		END_IF	
     *)
	180:
		Seal2CylinderUp.i.ActiveIn:=TRUE;
		Seal2CylinderUp.i.ActiveOut:=FALSE;		
		Seal2CylinderDown.i.ActiveIn:=TRUE;
		Seal2CylinderDown.i.ActiveOut:=FALSE;
		IF Seal2CylinderDown.i.InSensor AND Seal2CylinderUp.i.InSensor 
		AND NOT Seal2CylinderDown.o.Error 
		AND NOT Seal2CylinderUp.o.Error THEN
			Seal2Seq(Execute:= TRUE, Next:= 190); 
		END_IF
	
	190:
		  glb_Un01Box.Box[HMI_Seal2No].Seal2:=FALSE;
		  Seal2Seq(Execute:= TRUE,Hold:=FALSE, Next:= 110); 
	 
	Seq_StoppingDone:
		 IF  NOT Ref_MachineStateModel.Sts_Stopping THEN
			 Seal2Seq(Execute:= TRUE, Next:= 0); 
		 END_IF		 
 
END_CASE
Seal2Seq.Hold := Ref_MachineStateModel.Sts_Held;;
END_ACTION

ACTION CM08_Check1:
CASE Check1Seq.Now OF	
	0:
	   IF Ref_MachineStateModel.Sts_Execute  THEN
		  Check1Seq(Execute:= TRUE, Next:= 110);  
	   END_IF	
	
	   IF Ref_MachineStateModel.Sts_Stopping THEN
		  Check1Seq(Execute:= TRUE, Next:= Seq_StoppingDone);     
	   END_IF	
	
	110: 
		IF glb_Un01Box.Box[HMI_Check1No].Check1 THEN
		   Check1Seq(Execute:= TRUE, Next:= 120); 
		END_IF
		IF Ref_MachineStateModel.Sts_Stopping THEN
		   Check1Seq(Execute:= TRUE, Next:= Seq_StoppingDone);  
		END_IF	
		
	120: 
	    Check1Cylinder.i.ActiveIn:=FALSE;
		Check1Cylinder.i.ActiveOut:=TRUE;
		IF  Check1Cylinder.i.OutSensor AND NOT Check1Cylinder.o.Error  THEN
		 	Check1Seq(Execute:= TRUE, Next:= 121); 
		END_IF	  
		
	121:
		tonCheck1Seq(IN:=TRUE , PT:=T#2S , Q=> , ET=> );
		IF tonCheck1Seq.Q THEN
			tonCheck1Seq(IN:=FALSE , PT:=T#2S , Q=> , ET=> );
			Check1Seq(Execute:= TRUE,Hold:=FALSE, Next:= 130); 
		END_IF	
 
	130:
	    IF NOT check1Sensor1.o.Value THEN
           HMI_StopEvent[5].ID[20]:=TRUE;
		END_IF
	    IF NOT check1Sensor2.o.Value THEN
           HMI_StopEvent[5].ID[21]:=TRUE;
		END_IF
   	    IF NOT check1Sensor3.o.Value THEN
           HMI_StopEvent[5].ID[22]:=TRUE;
		END_IF
   	    IF NOT check1Sensor4.o.Value THEN
           HMI_StopEvent[5].ID[23]:=TRUE;
		END_IF
   	    IF NOT check1Sensor5.o.Value THEN
           HMI_StopEvent[5].ID[24]:=TRUE;
		END_IF
   	    IF NOT check1Sensor6.o.Value THEN
           HMI_StopEvent[5].ID[25]:=TRUE;
		END_IF
   	    IF NOT check1Sensor7.o.Value THEN
           HMI_StopEvent[5].ID[26]:=TRUE;
		END_IF
	    Check1Seq(Execute:= TRUE,Hold:=FALSE, Next:= 140);

  	  
	140:
		Check1Cylinder.i.ActiveIn:=TRUE;
		Check1Cylinder.i.ActiveOut:=FALSE;	
		IF  Check1Cylinder.i.InSensor AND NOT Check1Cylinder.o.Error  THEN
		    glb_Un01Box.Box[HMI_Check1No].Check1:=FALSE;
	        Check1Seq(Execute:= TRUE,Hold:=FALSE, Next:= 110); 
	     END_IF
		 
	Seq_StoppingDone:
		 IF  NOT Ref_MachineStateModel.Sts_Stopping THEN
			 Check1Seq(Execute:= TRUE, Next:= 0); 
		 END_IF		 
END_CASE
Check1Seq.Hold := Ref_MachineStateModel.Sts_Held;;
END_ACTION

ACTION CM09_Check2_Reject:
CASE RejectSeq.Now OF	
	0:
	   IF Ref_MachineStateModel.Sts_Execute  THEN
		  RejectSeq(Execute:= TRUE, Next:= 110);  
	   END_IF	
	
	   IF Ref_MachineStateModel.Sts_Stopping THEN
		  RejectSeq(Execute:= TRUE, Next:= Seq_StoppingDone);     
	   END_IF	
	
	110: 
		IF bRejectActive THEN
		   RejectSeq(Execute:= TRUE, Next:= 120); 
		END_IF
		IF Ref_MachineStateModel.Sts_Stopping THEN
		   RejectSeq(Execute:= TRUE, Next:= Seq_StoppingDone);  
		END_IF	
		
	120: 
	    RejectCylinder.i.ActiveIn:=FALSE;
		RejectCylinder.i.ActiveOut:=TRUE;
		IF  RejectCylinder.i.OutSensor AND NOT RejectCylinder.o.Error  THEN
		 	RejectSeq(Execute:= TRUE, Next:= 121); 
		END_IF	  
		
	121:
		tonRejectSeq(IN:=TRUE , PT:=T#1.5S , Q=> , ET=> );
		IF tonRejectSeq.Q THEN
			tonRejectSeq(IN:=FALSE , PT:=T#1.5S , Q=> , ET=> );
			RejectSeq(Execute:= TRUE,Hold:=FALSE, Next:= 130); 
		END_IF	
 
	130:
		RejectCylinder.i.ActiveIn:=TRUE;
		RejectCylinder.i.ActiveOut:=FALSE;	
		IF  RejectCylinder.i.InSensor AND NOT RejectCylinder.o.Error  THEN
		    bRejectActive:=FALSE;
	        RejectSeq(Execute:= TRUE,Hold:=FALSE, Next:= 110); 
	     END_IF
		 
	Seq_StoppingDone:
		 IF  NOT Ref_MachineStateModel.Sts_Stopping THEN
			 RejectSeq(Execute:= TRUE, Next:= 0); 
		 END_IF		 
END_CASE
RejectSeq.Hold := Ref_MachineStateModel.Sts_Held;;
END_ACTION

METHOD HomeValve : BOOL
VAR_INPUT
END_VAR
	PullCylinder1.i.ActiveIn:=TRUE;
	PullCylinder1.i.ActiveOut:=FALSE;
	PullCylinder2.i.ActiveIn:=TRUE;
	PullCylinder2.i.ActiveOut:=FALSE;
	PullCylinder3.i.ActiveIn:=TRUE;
	PullCylinder3.i.ActiveOut:=FALSE;
	PullCylinder4.i.ActiveIn:=TRUE;
	PullCylinder4.i.ActiveOut:=FALSE;
	PullCylinder5.i.ActiveIn:=TRUE;
	PullCylinder5.i.ActiveOut:=FALSE;
	PullCylinder6.i.ActiveIn:=TRUE;
	PullCylinder6.i.ActiveOut:=FALSE;
	PullCylinder7.i.ActiveIn:=TRUE;
	PullCylinder7.i.ActiveOut:=FALSE;
	PullVacuum1.i.ActiveIN:=FALSE;
	PullVacuum2.i.ActiveIN:=FALSE;
	PullVacuum3.i.ActiveIN:=FALSE;
	PullVacuum4.i.ActiveIN:=FALSE;
	PullVacuum5.i.ActiveIN:=FALSE;
	PullVacuum6.i.ActiveIN:=FALSE;
	PullVacuum7.i.ActiveIN:=FALSE;
	
	DropCylinderUP.i.ActiveIn:=TRUE;
	DropCylinderUP.i.ActiveOut:=FALSE;		
	DropCylinderDown.i.ActiveIn:=TRUE;
	DropCylinderDown.i.ActiveOut:=FALSE;

    Check1Cylinder.i.ActiveIn:=TRUE;
	Check1Cylinder.i.ActiveOut:=FALSE;
 
	
	CutCylinderUp.i.ActiveIn:=TRUE;
	CutCylinderUp.i.ActiveOut:=FALSE;
	CutCylinderDown.i.ActiveIn:=TRUE;
	CutCylinderDown.i.ActiveOut:=FALSE;
	
	SealCylinderUp.i.ActiveIn:=TRUE;
	SealCylinderUp.i.ActiveOut:=FALSE;
	
	SealCylinderDown.i.ActiveIn:=TRUE;
	SealCylinderDown.i.ActiveOut:=FALSE;

	Seal2CylinderUp.i.ActiveIn:=TRUE;
	Seal2CylinderUp.i.ActiveOut:=FALSE;
	
	Seal2CylinderDown.i.ActiveIn:=TRUE;
	Seal2CylinderDown.i.ActiveOut:=FALSE;

	
	TransferCyliderVert.i.ActiveIn:=TRUE;
	TransferCyliderVert.i.ActiveOut:=FALSE;

    IF 	TransferCyliderVert.i.InSensor THEN
		TransferCyliderRota.i.ActiveIn:=TRUE;
		TransferCyliderRota.i.ActiveOut:=FALSE;	
        IF 	TransferCyliderRota.i.InSensor THEN
		    TransferCyliderHori.i.ActiveIn:=TRUE;
		    TransferCyliderHori.i.ActiveOut:=FALSE;
        END_IF	
	END_IF

	TransferVacuum1.i.ActiveIN:=FALSE;
	TransferVacuum2.i.ActiveIN:=FALSE;
	TransferVacuum3.i.ActiveIN:=FALSE;
	TransferVacuum4.i.ActiveIN:=FALSE;
	TransferVacuum5.i.ActiveIN:=FALSE;
	TransferVacuum6.i.ActiveIN:=FALSE;
	TransferVacuum7.i.ActiveIN:=FALSE;	
    
HomeValve := PullCylinder1.i.InSensor AND NOT PullCylinder1.o.Error
AND PullCylinder2.i.InSensor AND NOT PullCylinder2.o.Error
AND PullCylinder3.i.InSensor AND NOT PullCylinder3.o.Error 
AND PullCylinder4.i.InSensor AND NOT PullCylinder4.o.Error 
AND PullCylinder5.i.InSensor AND NOT PullCylinder5.o.Error
AND PullCylinder6.i.InSensor AND NOT PullCylinder6.o.Error 
AND PullCylinder7.i.InSensor AND NOT PullCylinder7.o.Error
AND DropCylinderUP.i.InSensor AND Check1Cylinder.i.InSensor
AND  NOT Check1Cylinder.o.Error AND NOT DropCylinderUP.o.Error
AND DropCylinderDown.i.InSensor AND NOT DropCylinderDown.o.Error 
AND CutCylinderUp.i.InSensor AND NOT CutCylinderUp.o.Error 
AND CutCylinderDown.i.InSensor AND NOT CutCylinderDown.o.Error 
AND SealCylinderUp.i.InSensor AND NOT SealCylinderUp.o.Error 
AND SealCylinderDown.i.InSensor AND NOT SealCylinderDown.o.Error 
AND TransferCyliderHori.i.InSensor AND NOT TransferCyliderHori.o.Error
AND TransferCyliderRota.i.InSensor AND NOT TransferCyliderRota.o.Error 
AND TransferCyliderVert.i.InSensor AND NOT TransferCyliderVert.o.Error ;
END_METHOD

ACTION MainRoution:
EM_No:=7;
IF Ref_Unit.EM_Selected[EM_No] THEN
	IF Ref_MachineStateModel.Sts_Holding THEN
		Ref_Unit.EM_Holding_Done[EM_No]:=TRUE;
		ELSE
		Ref_Unit.EM_Holding_Done[EM_No]:=FALSE;
	END_IF
	IF Ref_MachineStateModel.Sts_UnHolding THEN
		Ref_Unit.EM_UnHolding_Done[EM_No]:=TRUE;
		ELSE
		Ref_Unit.EM_UnHolding_Done[EM_No]:=FALSE;
	END_IF
	
	IF Ref_MachineStateModel.Sts_Suspending THEN
		Ref_Unit.EM_Suspending_Done[EM_No]:=TRUE;
		ELSE
		Ref_Unit.EM_Suspending_Done[EM_No]:=FALSE;
	END_IF
	
	IF Ref_MachineStateModel.Sts_UnSuspending THEN
		Ref_Unit.EM_UnSuspending_Done[EM_No]:=TRUE;
		ELSE
		Ref_Unit.EM_UnSuspending_Done[EM_No]:=FALSE;
	END_IF
	

	IF Ref_MachineStateModel.Sts_Resetting AND beltSeq.Now=Seq_ResettingDone THEN
	   Ref_Unit.EM_Resetting_Done[EM_No]:=TRUE;
       ELSE   
	   Ref_Unit.EM_Resetting_Done[EM_No]:=FALSE;
	END_IF
	
	IF Ref_MachineStateModel.Sts_Clearing THEN
	   Ref_Unit.EM_Clearing_Done[EM_No]:=TRUE;  
    ELSE
	   Ref_Unit.EM_Clearing_Done[EM_No]:=FALSE;
	END_IF
	

	IF Ref_MachineStateModel.Sts_Starting THEN
	   Ref_Unit.EM_Starting_Done[EM_No]:=TRUE;
	ELSE
	   Ref_Unit.EM_Starting_Done[EM_No]:=FALSE;
	END_IF
	
	IF Ref_MachineStateModel.Sts_Stopping
    AND PullSeq.Now=Seq_StoppingDone
	AND DropSeq.Now=Seq_StoppingDone
	AND CutSeq.Now=Seq_StoppingDone
	AND SealSeq.Now=Seq_StoppingDone	
	AND TransferSeq.Now=Seq_StoppingDone
	AND BeltSeq.Now=Seq_StoppingDone THEN
	   Ref_Unit.EM_Stopping_Done[EM_No]:=TRUE;
	ELSE
	   Ref_Unit.EM_Stopping_Done[EM_No]:=FALSE;
	END_IF
		
	IF Ref_MachineStateModel.Sts_Aborting THEN
		PullSeq(ExeCute:= TRUE, Next:= 0);
		DropSeq(ExeCute:= TRUE, Next:= 0); 
		CutSeq(Execute:= TRUE, Next:= 0); 
		SealSeq(Execute:= TRUE, Next:= 0); 	
		Seal2Seq(Execute:= TRUE, Next:= 0); 			
		TransferSeq(ExeCute:= TRUE, Next:= 0);
		BeltSeq(Execute:= TRUE, Next:= 0);
	    Check1Seq(Execute:= TRUE, Next:= 0);	
        RejectSeq(Execute:= TRUE, Next:= 0);	
        IF ref_Belt.o.StandStill THEN
		   ref_Belt.i.Stop:=TRUE;
		END_IF
		IF ref_Puller.o.StandStill THEN
		   ref_Puller.i.Stop:=TRUE;
		END_IF		
        ReleaseValve();
		IF tonAbortingWatchDog.Q THEN 
		Ref_Unit.EM_Aborting_Done[EM_No]:=TRUE;
		ref_Belt.i.Disable:=TRUE;
		ref_Puller.i.Disable:=TRUE;	
		END_IF
	ELSE
	    Ref_Unit.EM_Aborting_Done[EM_No]:=FALSE;
	END_IF
	
	tonAbortingWatchDog(IN:= Ref_MachineStateModel.Sts_Aborting, PT:=T#3S , Q=> , ET=> );
	CM01_Pull();
	CM02_Drop();
	CM03_Cut();
	CM06_Seal();
    CM07_Seal2();	
	CM04_Transfer();
	CM08_Check1();
	CM09_check2_Reject();
	CM05_Belt();
	ELSE
	PullSeq(ExeCute:= TRUE, Next:= 0);
	DropSeq(ExeCute:= TRUE, Next:= 0); 
	CutSeq(Execute:= TRUE, Next:= 0); 
	SealSeq(Execute:= TRUE, Next:= 0); 
	Seal2Seq(Execute:= TRUE, Next:= 0);	
	TransferSeq(ExeCute:= TRUE, Next:= 0);
	BeltSeq(Execute:= TRUE, Next:= 0);
	Check1Seq(Execute:= TRUE, Next:= 0);
	RejectSeq(Execute:= TRUE, Next:= 0);
END_IF
END_ACTION

METHOD ReleaseValve : BOOL
VAR_INPUT
END_VAR
	PullCylinder1.i.ActiveIn:=FALSE;
	PullCylinder1.i.ActiveOut:=FALSE;
	PullCylinder2.i.ActiveIn:=FALSE;
	PullCylinder2.i.ActiveOut:=FALSE;
	PullCylinder3.i.ActiveIn:=FALSE;
	PullCylinder3.i.ActiveOut:=FALSE;
	PullCylinder4.i.ActiveIn:=FALSE;
	PullCylinder4.i.ActiveOut:=FALSE;
	PullCylinder5.i.ActiveIn:=FALSE;
	PullCylinder5.i.ActiveOut:=FALSE;
	PullCylinder6.i.ActiveIn:=FALSE;
	PullCylinder6.i.ActiveOut:=FALSE;
	PullCylinder7.i.ActiveIn:=FALSE;
	PullCylinder7.i.ActiveOut:=FALSE;
	PullVacuum1.i.ActiveIN:=FALSE;
	PullVacuum2.i.ActiveIN:=FALSE;
	PullVacuum3.i.ActiveIN:=FALSE;
	PullVacuum4.i.ActiveIN:=FALSE;
	PullVacuum5.i.ActiveIN:=FALSE;
	PullVacuum6.i.ActiveIN:=FALSE;
	PullVacuum7.i.ActiveIN:=FALSE;
	DropCylinderUP.i.ActiveIn:=FALSE;
	DropCylinderUP.i.ActiveOut:=FALSE;		
	DropCylinderDown.i.ActiveIn:=FALSE;
	DropCylinderDown.i.ActiveOut:=FALSE;	
	CutCylinderUp.i.ActiveIn:=FALSE;
	CutCylinderUp.i.ActiveOut:=FALSE;
	CutCylinderDown.i.ActiveIn:=FALSE;
	CutCylinderDown.i.ActiveOut:=FALSE;
	
	SealCylinderUp.i.ActiveIn:=FALSE;
	SealCylinderUp.i.ActiveOut:=FALSE;
	SealCylinderDown.i.ActiveIn:=FALSE;
	SealCylinderDown.i.ActiveOut:=FALSE;	
	
	Seal2CylinderUp.i.ActiveIn:=FALSE;
	Seal2CylinderUp.i.ActiveOut:=FALSE;
	Seal2CylinderDown.i.ActiveIn:=FALSE;
	Seal2CylinderDown.i.ActiveOut:=FALSE;	
	
	TransferCyliderHori.i.ActiveIn:=FALSE;
	TransferCyliderHori.i.ActiveOut:=FALSE;
	TransferCyliderRota.i.ActiveIn:=FALSE;
	TransferCyliderRota.i.ActiveOut:=FALSE;	
	TransferCyliderVert.i.ActiveIn:=FALSE;
	TransferCyliderVert.i.ActiveOut:=FALSE;
	TransferVacuum1.i.ActiveIN:=FALSE;
	TransferVacuum2.i.ActiveIN:=FALSE;
	TransferVacuum3.i.ActiveIN:=FALSE;
	TransferVacuum4.i.ActiveIN:=FALSE;
	TransferVacuum5.i.ActiveIN:=FALSE;
	TransferVacuum6.i.ActiveIN:=FALSE;
	TransferVacuum7.i.ActiveIN:=FALSE;
    infeedCylinder.i.ActiveIn:=FALSE;
	InfeedCylinder.i.ActiveOut:=FALSE;	
	ReleaseValve:=TRUE;
END_METHOD

ACTION SR999_FaultHandler:
;
END_ACTION

END_PROGRAM

// ---- POUs/PackMaL_UN01/EM08_Belt7.TcPOU
PROGRAM EM08_Belt7
VAR
	Ref_Belt: REFERENCE TO UDT_AXISADMIN;
	Ref_MachineStateModel: REFERENCE TO PackMlv3_StateModel;
	Ref_Unit: REFERENCE TO UDT_UnitAdmin;	
	ref_diTransferPick:REFERENCE TO DINT;
	ref_diPrint:REFERENCE TO DINT;
	ref_bTransferPut:REFERENCE TO bool;
	Ref_Robot: REFERENCE TO UDT_Scara;
	
	EM_No: INT:=8;
	tonAbortingWatchDog: TON;
	
	lrPosCnt: LREAL;
	tonBeltSeq: TON;
	Belt7Seq: SequenceTransfer;

	iBox: INT;
END_VAR

VAR CONSTANT
		
END_VAR
VAR RETAIN

END_VAR

//减速比25/1 同步轮周长40*10=400，皮带总长645*10= 6450，43个工位，工位间距150
Ref_MachineStateModel REF= UN01_MachineStateModel;
Ref_Unit REF=Unit01;
Ref_Belt REF= arRealAxisAdmin[48];
ref_diTransferPick REF= glb_diTransferPick_UN02;
ref_diPrint REF= glb_diPrint_UN02;
ref_bTransferPut REF= glb_bTransferPut_UN02;

MainRoution();
SR999_Faulthandler();

glb_bUnit02BoxEmpty:=NOT glb_Un02Box.Box[0].Valid 
AND NOT glb_Un02Box.Box[1].Valid AND NOT glb_Un02Box.Box[2].Valid AND NOT glb_Un02Box.Box[3].Valid 
AND NOT glb_Un02Box.Box[4].Valid AND NOT glb_Un02Box.Box[5].Valid AND NOT glb_Un02Box.Box[6].Valid 
AND NOT glb_Un02Box.Box[7].Valid AND NOT glb_Un02Box.Box[8].Valid AND NOT glb_Un02Box.Box[9].Valid 
AND NOT glb_Un02Box.Box[10].Valid AND NOT glb_Un02Box.Box[11].Valid AND NOT glb_Un02Box.Box[12].Valid 
AND NOT glb_Un02Box.Box[13].Valid AND NOT glb_Un02Box.Box[14].Valid AND NOT glb_Un02Box.Box[15].Valid 
AND NOT glb_Un02Box.Box[16].Valid AND NOT glb_Un02Box.Box[17].Valid AND NOT glb_Un02Box.Box[18].Valid 
AND NOT glb_Un02Box.Box[19].Valid AND NOT glb_Un02Box.Box[20].Valid AND NOT glb_Un02Box.Box[21].Valid ;

ACTION CM02_Belt:
  CASE Belt7Seq.Now  OF
	0: 
       IF Ref_MachineStateModel.Sts_Resetting THEN
		  Belt7Seq(Execute:= TRUE, Next:= Seq_Resetting);
	   END_IF	
       IF Ref_MachineStateModel.Sts_Execute THEN
		  Belt7Seq(Execute:= TRUE, Next:= 110);
	   END_IF
	   IF Ref_MachineStateModel.Sts_Stopping  THEN
		  Belt7Seq(Execute:= TRUE, Next:= Seq_Stopping);   
	   END_IF	


	   
	Seq_Resetting:
		IF NOT Ref_Belt.o.PowerOn  THEN;
		   Ref_Belt.i.Enable:=TRUE;
		ELSE
		   Belt7Seq(Execute:= TRUE, Next:= 20);  
		END_IF
		IF Ref_MachineStateModel.Sts_Stopping  THEN
		   Belt7Seq(Execute:= TRUE, Next:= Seq_Stopping);   
		END_IF		
		
	20:
	   IF NOT glb_AllAxisHomed_UN01 THEN
		  Belt7Seq(Execute:= TRUE, Next:= 21);   
		  ELSE
	      Belt7Seq(Execute:= TRUE, Next:= 30);  
	   END_IF
	   
	21: 
       MEMSET(destAddr:= ADR(glb_Un02Box), fillByte:= 0, n:= SIZEOF(glb_Un02Box));
       ref_diPrint:=0;
       Belt7Seq(Execute:= TRUE, Next:= 22); 
	   
	22:	
	   Ref_Belt.i.Home:=TRUE;
	   IF Ref_Belt.o.HomeDone THEN
		   Ref_Belt.i.Home:=FALSE;
		   Belt7Seq(Execute:= TRUE, Next:= 25);   
	   ELSE IF Ref_MachineStateModel.Sts_Stopping  THEN
		       Belt7Seq(Execute:= TRUE, Next:= Seq_Stopping);   
		    END_IF	 		   
	   END_IF
	   
	25:
		Ref_Belt.i.Pos:=0;
	    lrPosCnt:=1;	
	    Belt7Seq(Execute:= TRUE,Hold:= FALSE, Next:= 30);  

		
	30:			
		tonBeltSeq(IN:= TRUE, PT:= T#1S, Q=> , ET=> );
		IF tonBeltSeq.Q THEN
			tonBeltSeq(IN:= FALSE, PT:= T#1S, Q=> , ET=> );
			Ref_Belt.i.MoveAbs:=TRUE;	
			Belt7Seq(Execute:= TRUE, Next:= 31);  	   
		END_IF
			
    31:	
		IF  Ref_Belt.o.CmdDone THEN
		    Ref_Belt.i.MoveAbs:=FALSE;
            Belt7Seq(Execute:= TRUE, Next:= Seq_ResettingDone);  	
        ELSE IF Ref_MachineStateModel.Sts_Stopping  THEN
		        Belt7Seq(Execute:= TRUE, Next:= Seq_Stopping);     
	         END_IF		
		END_IF
		
	Seq_ResettingDone:
         IF NOT Ref_MachineStateModel.Sts_Resetting THEN
            Belt7Seq(Execute:= TRUE, Next:= 0);
         END_IF  	      
	   
		
